LIN {X 0,Y 359.461,Z 488.763,A -85,B 0,C 180,E1 -13387.725,E2 -13387.725} C_VEL
LIN {X 0,Y 362.812,Z 518.592,A -85,B 0,C 180,E1 -13388.562,E2 -13388.562} C_VEL
LIN {X 0,Y 363.143,Z 524.633,A -85,B 0,C 180,E1 -13388.708,E2 -13388.708} C_VEL
LIN {X 0,Y 361.795,Z 606.537,A -85,B 0,C 180,E1 -13390.348,E2 -13390.348} C_VEL
LIN {X 0,Y 361.078,Z 619.618,A -85,B 0,C 180,E1 -13390.825,E2 -13390.825} C_VEL
LIN {X 0,Y 360.35,Z 632.194,A -85,B 0,C 180,E1 -13391.522,E2 -13391.522} C_VEL
LIN {X 0,Y 359.408,Z 643.388,A -85,B 0,C 180,E1 -13392.356,E2 -13392.356} C_VEL
LIN {X 0,Y 358.272,Z 654.913,A -85,B 0,C 180,E1 -13393.475,E2 -13393.475} C_VEL
LIN {X 0,Y 357.239,Z 665.304,A -85,B 0,C 180,E1 -13394.749,E2 -13394.749} C_VEL
LIN {X 0,Y 356.357,Z 673.723,A -85,B 0,C 180,E1 -13396.019,E2 -13396.019} C_VEL
LIN {X 0,Y 355.447,Z 681.49,A -85,B 0,C 180,E1 -13397.438,E2 -13397.438} C_VEL
LIN {X 0,Y 354.634,Z 689.051,A -85,B 0,C 180,E1 -13399.148,E2 -13399.148} C_VEL
LIN {X 0,Y 354.06,Z 695.119,A -85,B 0,C 180,E1 -13400.863,E2 -13400.863} C_VEL
LIN {X 0,Y 353.628,Z 699.908,A -85,B 0,C 180,E1 -13402.578,E2 -13402.578} C_VEL
LIN {X 0,Y 353.416,Z 703.562,A -85,B 0,C 180,E1 -13404.293,E2 -13404.293} C_VEL
LIN {X 0,Y 353.372,Z 705.445,A -85,B 0,C 180,E1 -13405.437,E2 -13405.437} C_VEL
LIN {X 0,Y 353.285,Z 706.865,A -85,B 0,C 180,E1 -13406.578,E2 -13406.578} C_VEL
LIN {X 0,Y 353.239,Z 708.477,A -85,B 0,C 180,E1 -13408.86,E2 -13408.86} C_VEL
LIN {X 0,Y 353.281,Z 708.695,A -85,B 0,C 180,E1 -13410,E2 -13410} C_VEL
LIN {X 0,Y 353.285,Z 708.473,A -85,B 0,C 180,E1 -13411.14,E2 -13411.14} C_VEL
LIN {X 0,Y 353.291,Z 706.855,A -85,B 0,C 180,E1 -13413.421,E2 -13413.421} C_VEL
LIN {X 0,Y 353.381,Z 705.429,A -85,B 0,C 180,E1 -13414.563,E2 -13414.563} C_VEL
LIN {X 0,Y 353.476,Z 702.599,A -85,B 0,C 180,E1 -13416.212,E2 -13416.212} C_VEL
LIN {X 0,Y 353.734,Z 698.435,A -85,B 0,C 180,E1 -13417.994,E2 -13417.994} C_VEL
LIN {X 0,Y 354.314,Z 692.219,A -85,B 0,C 180,E1 -13419.995,E2 -13419.995} C_VEL
LIN {X 0,Y 354.986,Z 685.433,A -85,B 0,C 180,E1 -13421.708,E2 -13421.708} C_VEL
LIN {X 0,Y 355.811,Z 678.485,A -85,B 0,C 180,E1 -13423.129,E2 -13423.129} C_VEL
LIN {X 0,Y 356.713,Z 670.085,A -85,B 0,C 180,E1 -13424.549,E2 -13424.549} C_VEL
LIN {X 0,Y 357.781,Z 659.681,A -85,B 0,C 180,E1 -13425.962,E2 -13425.962} C_VEL
LIN {X 0,Y 358.816,Z 649.368,A -85,B 0,C 180,E1 -13427.086,E2 -13427.086} C_VEL
LIN {X 0,Y 359.843,Z 638.003,A -85,B 0,C 180,E1 -13428.062,E2 -13428.062} C_VEL
LIN {X 0,Y 360.766,Z 624.933,A -85,B 0,C 180,E1 -13428.897,E2 -13428.897} C_VEL
LIN {X 0,Y 361.503,Z 612.616,A -85,B 0,C 180,E1 -13429.447,E2 -13429.447} C_VEL
LIN {X 0,Y 361.878,Z 602.647,A -85,B 0,C 180,E1 -13429.758,E2 -13429.758} C_VEL
LIN {X 0,Y 363.518,Z 587.437,A -85,B 0,C 180,E1 -13430.587,E2 -13430.587} C_VEL
LIN {X 0,Y 364.531,Z 572.35,A -85,B 0,C 180,E1 -13431.155,E2 -13431.155} C_VEL
LIN {X 0,Y 366.818,Z 522.316,A -85,B 0,C 180,E1 -13432.636,E2 -13432.636} C_VEL
LIN {X 0,Y 365.737,Z 500.479,A -85,B 0,C 180,E1 -13433.543,E2 -13433.543} C_VEL
LIN {X 0,Y 363.696,Z 482.777,A -85,B 0,C 180,E1 -13434.452,E2 -13434.452} C_VEL
LIN {X 0,Y 360.558,Z 464.171,A -85,B 0,C 180,E1 -13435.599,E2 -13435.599} C_VEL
LIN {X 0,Y 359.9,Z 460.319,A -85,B 0,C 180,E1 -13435.889,E2 -13435.889} C_VEL
LIN {X 0,Y 362.247,Z 444.845,A -85,B 0,C 180,E1 -13439.014,E2 -13439.014} C_VEL
LIN {X 0,Y 363.495,Z 437.862,A -85,B 0,C 180,E1 -13440.5,E2 -13440.5} C_VEL
LIN {X 0,Y 362.465,Z 431.346,A -85,B 0,C 180,E1 -13442.222,E2 -13442.222} C_VEL
LIN {X 0,Y 360.838,Z 424.073,A -85,B 0,C 180,E1 -13444.391,E2 -13444.391} C_VEL
LIN {X 0,Y 358.871,Z 416.962,A -85,B 0,C 180,E1 -13446.843,E2 -13446.843} C_VEL
LIN {X 0,Y 356.686,Z 409.94,A -85,B 0,C 180,E1 -13449.786,E2 -13449.786} C_VEL
LIN {X 0,Y 354.81,Z 404.374,A -85,B 0,C 180,E1 -13452.814,E2 -13452.814} C_VEL
LIN {X 0,Y 354.763,Z 404.295,A -85,B 0,C 180,E1 -13456.103,E2 -13456.103} C_VEL
LIN {X 0,Y 354.765,Z 404.295,A -85,B 0,C 180,E1 -13459.176,E2 -13459.176} C_VEL
LIN {X 0,Y 354.801,Z 404.288,A -85,B 0,C 180,E1 -13462.404,E2 -13462.404} C_VEL
LIN {X 0,Y 354.813,Z 404.29,A -85,B 0,C 180,E1 -13464.941,E2 -13464.941} C_VEL
LIN {X 0,Y 354.795,Z 404.292,A -85,B 0,C 180,E1 -13468.405,E2 -13468.405} C_VEL
LIN {X 0,Y 354.804,Z 404.289,A -85,B 0,C 180,E1 -13471.615,E2 -13471.615} C_VEL
LIN {X 0,Y 354.878,Z 404.452,A -85,B 0,C 180,E1 -13473.459,E2 -13473.459} C_VEL
LIN {X 0,Y 355.056,Z 405.311,A -85,B 0,C 180,E1 -13473.704,E2 -13473.704} C_VEL
LIN {X 0,Y 356.467,Z 407.983,A -85,B 0,C 180,E1 -13474.099,E2 -13474.099} C_VEL
LIN {X 0,Y 357.72,Z 409.436,A -85,B 0,C 180,E1 -13474.372,E2 -13474.372} C_VEL
LIN {X 0,Y 359.867,Z 412.919,A -85,B 0,C 180,E1 -13474.879,E2 -13474.879} C_VEL
LIN {X 0,Y 366.309,Z 424.138,A -85,B 0,C 180,E1 -13476.306,E2 -13476.306} C_VEL
LIN {X 0,Y 370.407,Z 432.325,A -85,B 0,C 180,E1 -13477.154,E2 -13477.154} C_VEL
LIN {X 0,Y 367.524,Z 483.674,A -85,B 0,C 180,E1 -13478.769,E2 -13478.769} C_VEL
LIN {X 0,Y 367.158,Z 500.037,A -85,B 0,C 180,E1 -13479.37,E2 -13479.37} C_VEL
LIN {X 0,Y 366.638,Z 513.137,A -85,B 0,C 180,E1 -13480.075,E2 -13480.075} C_VEL
LIN {X 0,Y 365.817,Z 525.138,A -85,B 0,C 180,E1 -13480.937,E2 -13480.937} C_VEL
LIN {X 0,Y 364.914,Z 535.852,A -85,B 0,C 180,E1 -13481.907,E2 -13481.907} C_VEL
LIN {X 0,Y 363.634,Z 546.798,A -85,B 0,C 180,E1 -13483.148,E2 -13483.148} C_VEL
LIN {X 0,Y 362.445,Z 556.55,A -85,B 0,C 180,E1 -13484.537,E2 -13484.537} C_VEL
LIN {X 0,Y 361.097,Z 565.838,A -85,B 0,C 180,E1 -13486.207,E2 -13486.207} C_VEL
LIN {X 0,Y 360.036,Z 572.192,A -85,B 0,C 180,E1 -13487.601,E2 -13487.601} C_VEL
LIN {X 0,Y 358.912,Z 578.359,A -85,B 0,C 180,E1 -13489.279,E2 -13489.279} C_VEL
LIN {X 0,Y 357.917,Z 583.167,A -85,B 0,C 180,E1 -13490.962,E2 -13490.962} C_VEL
LIN {X 0,Y 357.17,Z 586.752,A -85,B 0,C 180,E1 -13492.652,E2 -13492.652} C_VEL
LIN {X 0,Y 356.406,Z 589.291,A -85,B 0,C 180,E1 -13494.342,E2 -13494.342} C_VEL
LIN {X 0,Y 356.167,Z 590.371,A -85,B 0,C 180,E1 -13495.473,E2 -13495.473} C_VEL
LIN {X 0,Y 355.862,Z 591.054,A -85,B 0,C 180,E1 -13496.603,E2 -13496.603} C_VEL
LIN {X 0,Y 355.612,Z 591.321,A -85,B 0,C 180,E1 -13497.735,E2 -13497.735} C_VEL
LIN {X 0,Y 355.304,Z 591.132,A -85,B 0,C 180,E1 -13498.867,E2 -13498.867} C_VEL
LIN {X 0,Y 355.064,Z 590.518,A -85,B 0,C 180,E1 -13500,E2 -13500} C_VEL
LIN {X 0,Y 355.062,Z 589.461,A -85,B 0,C 180,E1 -13501.134,E2 -13501.134} C_VEL
LIN {X 0,Y 354.997,Z 587.96,A -85,B 0,C 180,E1 -13502.269,E2 -13502.269} C_VEL
LIN {X 0,Y 354.982,Z 584.874,A -85,B 0,C 180,E1 -13503.973,E2 -13503.973} C_VEL
LIN {X 0,Y 355.19,Z 580.69,A -85,B 0,C 180,E1 -13505.678,E2 -13505.678} C_VEL
LIN {X 0,Y 355.54,Z 574.295,A -85,B 0,C 180,E1 -13507.668,E2 -13507.668} C_VEL
LIN {X 0,Y 355.933,Z 567.286,A -85,B 0,C 180,E1 -13509.375,E2 -13509.375} C_VEL
LIN {X 0,Y 356.366,Z 558.555,A -85,B 0,C 180,E1 -13511.086,E2 -13511.086} C_VEL
LIN {X 0,Y 356.866,Z 549.666,A -85,B 0,C 180,E1 -13512.511,E2 -13512.511} C_VEL
LIN {X 0,Y 357.419,Z 538.714,A -85,B 0,C 180,E1 -13513.938,E2 -13513.938} C_VEL
LIN {X 0,Y 358.013,Z 527.922,A -85,B 0,C 180,E1 -13515.076,E2 -13515.076} C_VEL
LIN {X 0,Y 358.444,Z 515.746,A -85,B 0,C 180,E1 -13516.107,E2 -13516.107} C_VEL
LIN {X 0,Y 358.803,Z 502.919,A -85,B 0,C 180,E1 -13516.939,E2 -13516.939} C_VEL
LIN {X 0,Y 359.093,Z 490.116,A -85,B 0,C 180,E1 -13517.549,E2 -13517.549} C_VEL
LIN {X 0,Y 359.22,Z 473.341,A -85,B 0,C 180,E1 -13518.058,E2 -13518.058} C_VEL
LIN {X 0,Y 360.312,Z 421.7,A -85,B 0,C 180,E1 -13519.417,E2 -13519.417} C_VEL
LIN {X 0,Y 354.994,Z 405.051,A -85,B 0,C 180,E1 -13520.111,E2 -13520.111} C_VEL
LIN {X 0,Y 354.865,Z 404.333,A -85,B 0,C 180,E1 -13520.354,E2 -13520.354} C_VEL
LIN {X 0,Y 354.859,Z 404.284,A -85,B 0,C 180,E1 -13524.351,E2 -13524.351} C_VEL
LIN {X 0,Y 354.805,Z 404.274,A -85,B 0,C 180,E1 -13528.385,E2 -13528.385} C_VEL
LIN {X 0,Y 354.789,Z 404.289,A -85,B 0,C 180,E1 -13532.333,E2 -13532.333} C_VEL
LIN {X 0,Y 354.824,Z 404.285,A -85,B 0,C 180,E1 -13535.699,E2 -13535.699} C_VEL
LIN {X 0,Y 354.826,Z 404.286,A -85,B 0,C 180,E1 -13539.424,E2 -13539.424} C_VEL
LIN {X 0,Y 354.789,Z 404.287,A -85,B 0,C 180,E1 -13542.867,E2 -13542.867} C_VEL
LIN {X 0,Y 354.768,Z 404.291,A -85,B 0,C 180,E1 -13546.104,E2 -13546.104} C_VEL
LIN {X 0,Y 354.787,Z 404.294,A -85,B 0,C 180,E1 -13549.179,E2 -13549.179} C_VEL
LIN {X 0,Y 354.802,Z 404.275,A -85,B 0,C 180,E1 -13552.404,E2 -13552.404} C_VEL
LIN {X 0,Y 354.867,Z 404.473,A -85,B 0,C 180,E1 -13553.737,E2 -13553.737} C_VEL
LIN {X 0,Y 358.473,Z 416.958,A -85,B 0,C 180,E1 -13556.214,E2 -13556.214} C_VEL
LIN {X 0,Y 362.219,Z 432.037,A -85,B 0,C 180,E1 -13559.051,E2 -13559.051} C_VEL
LIN {X 0,Y 363.272,Z 437.662,A -85,B 0,C 180,E1 -13560.054,E2 -13560.054} C_VEL
LIN {X 0,Y 361.925,Z 456.618,A -85,B 0,C 180,E1 -13563.022,E2 -13563.022} C_VEL
LIN {X 0,Y 360.281,Z 480.837,A -85,B 0,C 180,E1 -13566.66,E2 -13566.66} C_VEL
LIN {X 0,Y 359.891,Z 488.076,A -85,B 0,C 180,E1 -13567.657,E2 -13567.657} C_VEL
LIN {X 0,Y 363.691,Z 514.331,A -85,B 0,C 180,E1 -13568.46,E2 -13568.46} C_VEL
LIN {X 0,Y 362.716,Z 576.614,A -85,B 0,C 180,E1 -13569.699,E2 -13569.699} C_VEL
LIN {X 0,Y 362.221,Z 601.278,A -85,B 0,C 180,E1 -13570.225,E2 -13570.225} C_VEL
LIN {X 0,Y 361.585,Z 613.984,A -85,B 0,C 180,E1 -13570.706,E2 -13570.706} C_VEL
LIN {X 0,Y 360.763,Z 627.4,A -85,B 0,C 180,E1 -13571.471,E2 -13571.471} C_VEL
LIN {X 0,Y 359.697,Z 639.089,A -85,B 0,C 180,E1 -13572.371,E2 -13572.371} C_VEL
LIN {X 0,Y 358.606,Z 650.259,A -85,B 0,C 180,E1 -13573.491,E2 -13573.491} C_VEL
LIN {X 0,Y 357.682,Z 660.097,A -85,B 0,C 180,E1 -13574.726,E2 -13574.726} C_VEL
LIN {X 0,Y 356.669,Z 668.662,A -85,B 0,C 180,E1 -13576.032,E2 -13576.032} C_VEL
LIN {X 0,Y 355.529,Z 677.663,A -85,B 0,C 180,E1 -13577.731,E2 -13577.731} C_VEL
LIN {X 0,Y 354.758,Z 684.885,A -85,B 0,C 180,E1 -13579.441,E2 -13579.441} C_VEL
LIN {X 0,Y 354.025,Z 691.514,A -85,B 0,C 180,E1 -13581.438,E2 -13581.438} C_VEL
LIN {X 0,Y 353.666,Z 695.868,A -85,B 0,C 180,E1 -13583.152,E2 -13583.152} C_VEL
LIN {X 0,Y 353.479,Z 698.16,A -85,B 0,C 180,E1 -13584.295,E2 -13584.295} C_VEL
LIN {X 0,Y 353.366,Z 700.029,A -85,B 0,C 180,E1 -13585.437,E2 -13585.437} C_VEL
LIN {X 0,Y 353.244,Z 701.457,A -85,B 0,C 180,E1 -13586.578,E2 -13586.578} C_VEL
LIN {X 0,Y 353.158,Z 703.075,A -85,B 0,C 180,E1 -13588.86,E2 -13588.86} C_VEL
LIN {X 0,Y 353.175,Z 703.31,A -85,B 0,C 180,E1 -13590,E2 -13590} C_VEL
LIN {X 0,Y 353.158,Z 703.117,A -85,B 0,C 180,E1 -13591.14,E2 -13591.14} C_VEL
LIN {X 0,Y 353.243,Z 701.554,A -85,B 0,C 180,E1 -13593.422,E2 -13593.422} C_VEL
LIN {X 0,Y 353.36,Z 700.18,A -85,B 0,C 180,E1 -13594.563,E2 -13594.563} C_VEL
LIN {X 0,Y 353.525,Z 697.282,A -85,B 0,C 180,E1 -13596.283,E2 -13596.283} C_VEL
LIN {X 0,Y 353.823,Z 693.372,A -85,B 0,C 180,E1 -13597.993,E2 -13597.993} C_VEL
LIN {X 0,Y 354.368,Z 688.291,A -85,B 0,C 180,E1 -13599.705,E2 -13599.705} C_VEL
LIN {X 0,Y 355.088,Z 681.888,A -85,B 0,C 180,E1 -13601.416,E2 -13601.416} C_VEL
LIN {X 0,Y 355.944,Z 674.557,A -85,B 0,C 180,E1 -13603,E2 -13603} C_VEL
LIN {X 0,Y 355.766,Z 670.779,A -85,B 0,C 180,E1 -13603.732,E2 -13603.732} C_VEL
LIN {X 0,Y 353.689,Z 664.355,A -85,B 0,C 180,E1 -13604.912,E2 -13604.912} C_VEL
LIN {X 0,Y 351.651,Z 657.479,A -85,B 0,C 180,E1 -13606.029,E2 -13606.029} C_VEL
LIN {X 0,Y 351.516,Z 652.894,A -85,B 0,C 180,E1 -13606.642,E2 -13606.642} C_VEL
LIN {X 0,Y 352.757,Z 641.711,A -85,B 0,C 180,E1 -13607.838,E2 -13607.838} C_VEL
LIN {X 0,Y 353.851,Z 629.822,A -85,B 0,C 180,E1 -13608.83,E2 -13608.83} C_VEL
LIN {X 0,Y 354.693,Z 617.392,A -85,B 0,C 180,E1 -13609.61,E2 -13609.61} C_VEL
LIN {X 0,Y 355.48,Z 604.249,A -85,B 0,C 180,E1 -13610.167,E2 -13610.167} C_VEL
LIN {X 0,Y 355.953,Z 590.394,A -85,B 0,C 180,E1 -13610.516,E2 -13610.516} C_VEL
LIN {X 0,Y 357.122,Z 514.751,A -85,B 0,C 180,E1 -13612.052,E2 -13612.052} C_VEL
LIN {X 0,Y 353.268,Z 487.892,A -85,B 0,C 180,E1 -13612.904,E2 -13612.904} C_VEL
LIN {X 0,Y 354.289,Z 470.851,A -85,B 0,C 180,E1 -13615.403,E2 -13615.403} C_VEL
LIN {X 0,Y 356.179,Z 446.213,A -85,B 0,C 180,E1 -13619.233,E2 -13619.233} C_VEL
LIN {X 0,Y 356.668,Z 440.12,A -85,B 0,C 180,E1 -13620.201,E2 -13620.201} C_VEL
LIN {X 0,Y 354.578,Z 429.7,A -85,B 0,C 180,E1 -13622.125,E2 -13622.125} C_VEL
LIN {X 0,Y 350.938,Z 415.804,A -85,B 0,C 180,E1 -13624.807,E2 -13624.807} C_VEL
LIN {X 0,Y 347.815,Z 405.367,A -85,B 0,C 180,E1 -13626.938,E2 -13626.938} C_VEL
LIN {X 0,Y 347.699,Z 405.157,A -85,B 0,C 180,E1 -13630.302,E2 -13630.302} C_VEL
LIN {X 0,Y 347.723,Z 405.159,A -85,B 0,C 180,E1 -13633.409,E2 -13633.409} C_VEL
LIN {X 0,Y 347.727,Z 405.168,A -85,B 0,C 180,E1 -13636.687,E2 -13636.687} C_VEL
LIN {X 0,Y 347.703,Z 405.174,A -85,B 0,C 180,E1 -13640.182,E2 -13640.182} C_VEL
LIN {X 0,Y 347.757,Z 405.157,A -85,B 0,C 180,E1 -13642.678,E2 -13642.678} C_VEL
LIN {X 0,Y 347.751,Z 405.158,A -85,B 0,C 180,E1 -13645.956,E2 -13645.956} C_VEL
LIN {X 0,Y 347.741,Z 405.167,A -85,B 0,C 180,E1 -13649.651,E2 -13649.651} C_VEL
LIN {X 0,Y 347.743,Z 405.172,A -85,B 0,C 180,E1 -13653.6,E2 -13653.6} C_VEL
LIN {X 0,Y 347.766,Z 405.15,A -85,B 0,C 180,E1 -13656.16,E2 -13656.16} C_VEL
LIN {X 0,Y 347.783,Z 405.162,A -85,B 0,C 180,E1 -13659.907,E2 -13659.907} C_VEL
LIN {X 0,Y 347.801,Z 405.15,A -85,B 0,C 180,E1 -13663.567,E2 -13663.567} C_VEL
LIN {X 0,Y 347.888,Z 405.141,A -85,B 0,C 180,E1 -13667.16,E2 -13667.16} C_VEL
LIN {X 0,Y 347.937,Z 405.139,A -85,B 0,C 180,E1 -13670.701,E2 -13670.701} C_VEL
LIN {X 0,Y 348.04,Z 405.116,A -85,B 0,C 180,E1 -13674.205,E2 -13674.205} C_VEL
LIN {X 0,Y 348.19,Z 405.107,A -85,B 0,C 180,E1 -13677.686,E2 -13677.686} C_VEL
LIN {X 0,Y 348.119,Z 405.109,A -85,B 0,C 180,E1 -13681.157,E2 -13681.157} C_VEL
LIN {X 0,Y 348.185,Z 405.089,A -85,B 0,C 180,E1 -13682.314,E2 -13682.314} C_VEL
LIN {X 0,Y 348.058,Z 405.127,A -85,B 0,C 180,E1 -13686.959,E2 -13686.959} C_VEL
LIN {X 0,Y 347.894,Z 405.132,A -85,B 0,C 180,E1 -13690.475,E2 -13690.475} C_VEL
LIN {X 0,Y 347.859,Z 405.15,A -85,B 0,C 180,E1 -13694.122,E2 -13694.122} C_VEL
LIN {X 0,Y 347.79,Z 405.155,A -85,B 0,C 180,E1 -13698.238,E2 -13698.238} C_VEL
LIN {X 0,Y 347.766,Z 405.156,A -85,B 0,C 180,E1 -13701.624,E2 -13701.624} C_VEL
LIN {X 0,Y 347.741,Z 405.164,A -85,B 0,C 180,E1 -13705.114,E2 -13705.114} C_VEL
LIN {X 0,Y 347.731,Z 405.161,A -85,B 0,C 180,E1 -13707.701,E2 -13707.701} C_VEL
LIN {X 0,Y 347.741,Z 405.162,A -85,B 0,C 180,E1 -13710.349,E2 -13710.349} C_VEL
LIN {X 0,Y 347.75,Z 405.154,A -85,B 0,C 180,E1 -13714.043,E2 -13714.043} C_VEL
LIN {X 0,Y 347.756,Z 405.168,A -85,B 0,C 180,E1 -13717.322,E2 -13717.322} C_VEL
LIN {X 0,Y 347.697,Z 405.133,A -85,B 0,C 180,E1 -13720.302,E2 -13720.302} C_VEL
LIN {X 0,Y 347.722,Z 405.148,A -85,B 0,C 180,E1 -13723.408,E2 -13723.408} C_VEL
LIN {X 0,Y 347.724,Z 405.164,A -85,B 0,C 180,E1 -13726.687,E2 -13726.687} C_VEL
LIN {X 0,Y 347.702,Z 405.145,A -85,B 0,C 180,E1 -13730.182,E2 -13730.182} C_VEL
LIN {X 0,Y 347.755,Z 405.168,A -85,B 0,C 180,E1 -13732.678,E2 -13732.678} C_VEL
LIN {X 0,Y 347.84,Z 405.386,A -85,B 0,C 180,E1 -13734.974,E2 -13734.974} C_VEL
LIN {X 0,Y 351.815,Z 423.417,A -85,B 0,C 180,E1 -13738.709,E2 -13738.709} C_VEL
LIN {X 0,Y 353.402,Z 430.82,A -85,B 0,C 180,E1 -13740.187,E2 -13740.187} C_VEL
LIN {X 0,Y 353.222,Z 435.729,A -85,B 0,C 180,E1 -13741.1,E2 -13741.1} C_VEL
LIN {X 0,Y 350.983,Z 459.339,A -85,B 0,C 180,E1 -13745.37,E2 -13745.37} C_VEL
LIN {X 0,Y 352.006,Z 474.914,A -85,B 0,C 180,E1 -13746.387,E2 -13746.387} C_VEL
LIN {X 0,Y 352.822,Z 488.798,A -85,B 0,C 180,E1 -13747.281,E2 -13747.281} C_VEL
LIN {X 0,Y 356.443,Z 521.377,A -85,B 0,C 180,E1 -13748.217,E2 -13748.217} C_VEL
LIN {X 0,Y 355.687,Z 575.748,A -85,B 0,C 180,E1 -13749.317,E2 -13749.317} C_VEL
LIN {X 0,Y 355.114,Z 606.569,A -85,B 0,C 180,E1 -13749.963,E2 -13749.963} C_VEL
LIN {X 0,Y 354.386,Z 619.613,A -85,B 0,C 180,E1 -13750.448,E2 -13750.448} C_VEL
LIN {X 0,Y 353.618,Z 632.173,A -85,B 0,C 180,E1 -13751.158,E2 -13751.158} C_VEL
LIN {X 0,Y 352.65,Z 643.356,A -85,B 0,C 180,E1 -13752.007,E2 -13752.007} C_VEL
LIN {X 0,Y 351.445,Z 654.875,A -85,B 0,C 180,E1 -13753.144,E2 -13753.144} C_VEL
LIN {X 0,Y 350.3,Z 665.989,A -85,B 0,C 180,E1 -13754.543,E2 -13754.543} C_VEL
LIN {X 0,Y 349.271,Z 675.329,A -85,B 0,C 180,E1 -13756.027,E2 -13756.027} C_VEL
LIN {X 0,Y 348.164,Z 684.141,A -85,B 0,C 180,E1 -13757.763,E2 -13757.763} C_VEL
LIN {X 0,Y 347.381,Z 691.2,A -85,B 0,C 180,E1 -13759.509,E2 -13759.509} C_VEL
LIN {X 0,Y 346.836,Z 696.808,A -85,B 0,C 180,E1 -13761.258,E2 -13761.258} C_VEL
LIN {X 0,Y 346.444,Z 701.198,A -85,B 0,C 180,E1 -13763.009,E2 -13763.009} C_VEL
LIN {X 0,Y 346.338,Z 703.51,A -85,B 0,C 180,E1 -13764.176,E2 -13764.176} C_VEL
LIN {X 0,Y 346.286,Z 705.392,A -85,B 0,C 180,E1 -13765.343,E2 -13765.343} C_VEL
LIN {X 0,Y 346.208,Z 706.811,A -85,B 0,C 180,E1 -13766.508,E2 -13766.508} C_VEL
LIN {X 0,Y 346.139,Z 708.424,A -85,B 0,C 180,E1 -13768.836,E2 -13768.836} C_VEL
LIN {X 0,Y 346.181,Z 708.641,A -85,B 0,C 180,E1 -13770,E2 -13770} C_VEL
LIN {X 0,Y 346.183,Z 708.419,A -85,B 0,C 180,E1 -13771.163,E2 -13771.163} C_VEL
LIN {X 0,Y 346.214,Z 706.801,A -85,B 0,C 180,E1 -13773.491,E2 -13773.491} C_VEL
LIN {X 0,Y 346.295,Z 705.375,A -85,B 0,C 180,E1 -13774.656,E2 -13774.656} C_VEL
LIN {X 0,Y 346.401,Z 702.799,A -85,B 0,C 180,E1 -13776.202,E2 -13776.202} C_VEL
LIN {X 0,Y 346.678,Z 698.38,A -85,B 0,C 180,E1 -13778.158,E2 -13778.158} C_VEL
LIN {X 0,Y 347.298,Z 692.166,A -85,B 0,C 180,E1 -13780.199,E2 -13780.199} C_VEL
LIN {X 0,Y 348.018,Z 685.381,A -85,B 0,C 180,E1 -13781.946,E2 -13781.946} C_VEL
LIN {X 0,Y 348.869,Z 678.434,A -85,B 0,C 180,E1 -13783.395,E2 -13783.395} C_VEL
LIN {X 0,Y 349.813,Z 670.035,A -85,B 0,C 180,E1 -13784.842,E2 -13784.842} C_VEL
LIN {X 0,Y 350.935,Z 659.634,A -85,B 0,C 180,E1 -13786.282,E2 -13786.282} C_VEL
LIN {X 0,Y 352.017,Z 649.324,A -85,B 0,C 180,E1 -13787.426,E2 -13787.426} C_VEL
LIN {X 0,Y 353.111,Z 637.965,A -85,B 0,C 180,E1 -13788.419,E2 -13788.419} C_VEL
LIN {X 0,Y 354.073,Z 624.904,A -85,B 0,C 180,E1 -13789.268,E2 -13789.268} C_VEL
LIN {X 0,Y 354.815,Z 612.603,A -85,B 0,C 180,E1 -13789.828,E2 -13789.828} C_VEL
LIN {X 0,Y 355.175,Z 604.546,A -85,B 0,C 180,E1 -13790.109,E2 -13790.109} C_VEL
LIN {X 0,Y 356.965,Z 589.971,A -85,B 0,C 180,E1 -13790.982,E2 -13790.982} C_VEL
LIN {X 0,Y 358.206,Z 575.233,A -85,B 0,C 180,E1 -13791.622,E2 -13791.622} C_VEL
LIN {X 0,Y 360.877,Z 523.641,A -85,B 0,C 180,E1 -13793.205,E2 -13793.205} C_VEL
LIN {X 0,Y 359.91,Z 501.776,A -85,B 0,C 180,E1 -13794.15,E2 -13794.15} C_VEL
LIN {X 0,Y 358.015,Z 484.588,A -85,B 0,C 180,E1 -13795.074,E2 -13795.074} C_VEL
LIN {X 0,Y 355.218,Z 467.047,A -85,B 0,C 180,E1 -13796.191,E2 -13796.191} C_VEL
LIN {X 0,Y 353.681,Z 458.471,A -85,B 0,C 180,E1 -13796.837,E2 -13796.837} C_VEL
LIN {X 0,Y 356.403,Z 442.572,A -85,B 0,C 180,E1 -13800.188,E2 -13800.188} C_VEL
LIN {X 0,Y 356.899,Z 439.821,A -85,B 0,C 180,E1 -13800.796,E2 -13800.796} C_VEL
LIN {X 0,Y 355.608,Z 432.185,A -85,B 0,C 180,E1 -13802.922,E2 -13802.922} C_VEL
LIN {X 0,Y 353.753,Z 424.318,A -85,B 0,C 180,E1 -13805.457,E2 -13805.457} C_VEL
LIN {X 0,Y 352.199,Z 418.863,A -85,B 0,C 180,E1 -13807.498,E2 -13807.498} C_VEL
LIN {X 0,Y 350.206,Z 412.597,A -85,B 0,C 180,E1 -13810.307,E2 -13810.307} C_VEL
LIN {X 0,Y 348.392,Z 407.393,A -85,B 0,C 180,E1 -13813.304,E2 -13813.304} C_VEL
LIN {X 0,Y 347.704,Z 405.199,A -85,B 0,C 180,E1 -13815.027,E2 -13815.027} C_VEL
LIN {X 0,Y 347.74,Z 405.167,A -85,B 0,C 180,E1 -13818.399,E2 -13818.399} C_VEL
LIN {X 0,Y 347.757,Z 405.167,A -85,B 0,C 180,E1 -13822.678,E2 -13822.678} C_VEL
LIN {X 0,Y 347.749,Z 405.166,A -85,B 0,C 180,E1 -13825.956,E2 -13825.956} C_VEL
LIN {X 0,Y 347.742,Z 405.168,A -85,B 0,C 180,E1 -13829.651,E2 -13829.651} C_VEL
LIN {X 0,Y 347.797,Z 405.409,A -85,B 0,C 180,E1 -13832.223,E2 -13832.223} C_VEL
LIN {X 0,Y 347.973,Z 406.187,A -85,B 0,C 180,E1 -13832.441,E2 -13832.441} C_VEL
LIN {X 0,Y 349.437,Z 408.915,A -85,B 0,C 180,E1 -13832.889,E2 -13832.889} C_VEL
LIN {X 0,Y 351.057,Z 410.737,A -85,B 0,C 180,E1 -13833.29,E2 -13833.29} C_VEL
LIN {X 0,Y 353.011,Z 413.918,A -85,B 0,C 180,E1 -13833.818,E2 -13833.818} C_VEL
LIN {X 0,Y 358.572,Z 423.002,A -85,B 0,C 180,E1 -13835.153,E2 -13835.153} C_VEL
LIN {X 0,Y 364.152,Z 433.748,A -85,B 0,C 180,E1 -13836.426,E2 -13836.426} C_VEL
LIN {X 0,Y 364.737,Z 435.343,A -85,B 0,C 180,E1 -13836.567,E2 -13836.567} C_VEL
LIN {X 0,Y 361.707,Z 483.693,A -85,B 0,C 180,E1 -13838.123,E2 -13838.123} C_VEL
LIN {X 0,Y 361.209,Z 501.37,A -85,B 0,C 180,E1 -13838.798,E2 -13838.798} C_VEL
LIN {X 0,Y 360.699,Z 513.766,A -85,B 0,C 180,E1 -13839.469,E2 -13839.469} C_VEL
LIN {X 0,Y 359.898,Z 524.737,A -85,B 0,C 180,E1 -13840.247,E2 -13840.247} C_VEL
LIN {X 0,Y 358.866,Z 536.261,A -85,B 0,C 180,E1 -13841.296,E2 -13841.296} C_VEL
LIN {X 0,Y 357.483,Z 547.309,A -85,B 0,C 180,E1 -13842.554,E2 -13842.554} C_VEL
LIN {X 0,Y 356.203,Z 557.181,A -85,B 0,C 180,E1 -13843.965,E2 -13843.965} C_VEL
LIN {X 0,Y 354.989,Z 565.242,A -85,B 0,C 180,E1 -13845.379,E2 -13845.379} C_VEL
LIN {X 0,Y 353.608,Z 572.804,A -85,B 0,C 180,E1 -13847.021,E2 -13847.021} C_VEL
LIN {X 0,Y 352.559,Z 578.282,A -85,B 0,C 180,E1 -13848.502,E2 -13848.502} C_VEL
LIN {X 0,Y 351.488,Z 583.348,A -85,B 0,C 180,E1 -13850.215,E2 -13850.215} C_VEL
LIN {X 0,Y 350.469,Z 587.238,A -85,B 0,C 180,E1 -13851.931,E2 -13851.931} C_VEL
LIN {X 0,Y 349.925,Z 589.217,A -85,B 0,C 180,E1 -13853.079,E2 -13853.079} C_VEL
LIN {X 0,Y 349.498,Z 590.68,A -85,B 0,C 180,E1 -13854.23,E2 -13854.23} C_VEL
LIN {X 0,Y 349.232,Z 591.682,A -85,B 0,C 180,E1 -13855.383,E2 -13855.383} C_VEL
LIN {X 0,Y 348.885,Z 592.298,A -85,B 0,C 180,E1 -13856.535,E2 -13856.535} C_VEL
LIN {X 0,Y 348.619,Z 592.461,A -85,B 0,C 180,E1 -13857.689,E2 -13857.689} C_VEL
LIN {X 0,Y 348.294,Z 592.197,A -85,B 0,C 180,E1 -13858.844,E2 -13858.844} C_VEL
LIN {X 0,Y 348.036,Z 591.518,A -85,B 0,C 180,E1 -13860,E2 -13860} C_VEL
LIN {X 0,Y 348.036,Z 590.378,A -85,B 0,C 180,E1 -13861.157,E2 -13861.157} C_VEL
LIN {X 0,Y 347.965,Z 587.843,A -85,B 0,C 180,E1 -13862.894,E2 -13862.894} C_VEL
LIN {X 0,Y 347.885,Z 584.272,A -85,B 0,C 180,E1 -13864.635,E2 -13864.635} C_VEL
LIN {X 0,Y 348.277,Z 579.533,A -85,B 0,C 180,E1 -13866.372,E2 -13866.372} C_VEL
LIN {X 0,Y 348.571,Z 573.545,A -85,B 0,C 180,E1 -13868.114,E2 -13868.114} C_VEL
LIN {X 0,Y 348.975,Z 566.105,A -85,B 0,C 180,E1 -13869.857,E2 -13869.857} C_VEL
LIN {X 0,Y 349.39,Z 558.54,A -85,B 0,C 180,E1 -13871.31,E2 -13871.31} C_VEL
LIN {X 0,Y 349.926,Z 548.358,A -85,B 0,C 180,E1 -13872.911,E2 -13872.911} C_VEL
LIN {X 0,Y 350.537,Z 536.912,A -85,B 0,C 180,E1 -13874.366,E2 -13874.366} C_VEL
LIN {X 0,Y 351.172,Z 525.512,A -85,B 0,C 180,E1 -13875.514,E2 -13875.514} C_VEL
LIN {X 0,Y 351.599,Z 512.622,A -85,B 0,C 180,E1 -13876.549,E2 -13876.549} C_VEL
LIN {X 0,Y 351.962,Z 499.83,A -85,B 0,C 180,E1 -13877.316,E2 -13877.316} C_VEL
LIN {X 0,Y 352.202,Z 486.115,A -85,B 0,C 180,E1 -13877.904,E2 -13877.904} C_VEL
LIN {X 0,Y 352.864,Z 445.943,A -85,B 0,C 180,E1 -13879,E2 -13879} C_VEL
LIN {X 0,Y 353.285,Z 422.754,A -85,B 0,C 180,E1 -13879.64,E2 -13879.64} C_VEL
LIN {X 0,Y 348.008,Z 406.168,A -85,B 0,C 180,E1 -13880.331,E2 -13880.331} C_VEL
LIN {X 0,Y 347.826,Z 405.249,A -85,B 0,C 180,E1 -13880.552,E2 -13880.552} C_VEL
LIN {X 0,Y 347.813,Z 405.162,A -85,B 0,C 180,E1 -13884.593,E2 -13884.593} C_VEL
LIN {X 0,Y 347.743,Z 405.159,A -85,B 0,C 180,E1 -13887.7,E2 -13887.7} C_VEL
LIN {X 0,Y 347.743,Z 405.163,A -85,B 0,C 180,E1 -13890.349,E2 -13890.349} C_VEL
LIN {X 0,Y 347.75,Z 405.152,A -85,B 0,C 180,E1 -13894.044,E2 -13894.044} C_VEL
LIN {X 0,Y 347.763,Z 405.16,A -85,B 0,C 180,E1 -13897.321,E2 -13897.321} C_VEL
LIN {X 0,Y 347.734,Z 405.172,A -85,B 0,C 180,E1 -13900.297,E2 -13900.297} C_VEL
LIN {X 0,Y 347.725,Z 405.172,A -85,B 0,C 180,E1 -13903.408,E2 -13903.408} C_VEL
LIN {X 0,Y 347.727,Z 405.173,A -85,B 0,C 180,E1 -13906.686,E2 -13906.686} C_VEL
LIN {X 0,Y 347.73,Z 405.159,A -85,B 0,C 180,E1 -13910.177,E2 -13910.177} C_VEL
LIN {X 0,Y 347.79,Z 405.363,A -85,B 0,C 180,E1 -13913.171,E2 -13913.171} C_VEL
LIN {X 0,Y 351.416,Z 417.393,A -85,B 0,C 180,E1 -13915.62,E2 -13915.62} C_VEL
LIN {X 0,Y 354.973,Z 431.63,A -85,B 0,C 180,E1 -13918.359,E2 -13918.359} C_VEL
LIN {X 0,Y 356.568,Z 439.347,A -85,B 0,C 180,E1 -13919.784,E2 -13919.784} C_VEL
LIN {X 0,Y 355.266,Z 457.299,A -85,B 0,C 180,E1 -13922.617,E2 -13922.617} C_VEL
LIN {X 0,Y 353.644,Z 480.117,A -85,B 0,C 180,E1 -13926.088,E2 -13926.088} C_VEL
LIN {X 0,Y 353.202,Z 488.114,A -85,B 0,C 180,E1 -13927.213,E2 -13927.213} C_VEL
LIN {X 0,Y 357.131,Z 515.394,A -85,B 0,C 180,E1 -13928.067,E2 -13928.067} C_VEL
LIN {X 0,Y 355.665,Z 598.661,A -85,B 0,C 180,E1 -13929.769,E2 -13929.769} C_VEL
LIN {X 0,Y 355.037,Z 611.718,A -85,B 0,C 180,E1 -13930.222,E2 -13930.222} C_VEL
LIN {X 0,Y 354.396,Z 623.121,A -85,B 0,C 180,E1 -13930.825,E2 -13930.825} C_VEL
LIN {X 0,Y 353.433,Z 634.124,A -85,B 0,C 180,E1 -13931.599,E2 -13931.599} C_VEL
LIN {X 0,Y 352.359,Z 645.038,A -85,B 0,C 180,E1 -13932.592,E2 -13932.592} C_VEL
LIN {X 0,Y 351.242,Z 655.794,A -85,B 0,C 180,E1 -13933.829,E2 -13933.829} C_VEL
LIN {X 0,Y 350.238,Z 665.225,A -85,B 0,C 180,E1 -13935.176,E2 -13935.176} C_VEL
LIN {X 0,Y 348.941,Z 674.928,A -85,B 0,C 180,E1 -13936.904,E2 -13936.904} C_VEL
LIN {X 0,Y 348.026,Z 682.727,A -85,B 0,C 180,E1 -13938.645,E2 -13938.645} C_VEL
LIN {X 0,Y 347.413,Z 687.998,A -85,B 0,C 180,E1 -13940.099,E2 -13940.099} C_VEL
LIN {X 0,Y 346.831,Z 693.15,A -85,B 0,C 180,E1 -13941.846,E2 -13941.846} C_VEL
LIN {X 0,Y 346.501,Z 697.248,A -85,B 0,C 180,E1 -13943.648,E2 -13943.648} C_VEL
LIN {X 0,Y 346.285,Z 700.083,A -85,B 0,C 180,E1 -13945.344,E2 -13945.344} C_VEL
LIN {X 0,Y 346.171,Z 701.511,A -85,B 0,C 180,E1 -13946.508,E2 -13946.508} C_VEL
LIN {X 0,Y 346.061,Z 703.129,A -85,B 0,C 180,E1 -13948.836,E2 -13948.836} C_VEL
LIN {X 0,Y 346.076,Z 703.364,A -85,B 0,C 180,E1 -13950,E2 -13950} C_VEL
LIN {X 0,Y 346.061,Z 703.171,A -85,B 0,C 180,E1 -13951.164,E2 -13951.164} C_VEL
LIN {X 0,Y 346.17,Z 701.607,A -85,B 0,C 180,E1 -13953.492,E2 -13953.492} C_VEL
LIN {X 0,Y 346.279,Z 700.233,A -85,B 0,C 180,E1 -13954.657,E2 -13954.657} C_VEL
LIN {X 0,Y 346.449,Z 697.588,A -85,B 0,C 180,E1 -13956.274,E2 -13956.274} C_VEL
LIN {X 0,Y 346.776,Z 693.424,A -85,B 0,C 180,E1 -13958.156,E2 -13958.156} C_VEL
LIN {X 0,Y 347.352,Z 688.342,A -85,B 0,C 180,E1 -13959.903,E2 -13959.903} C_VEL
LIN {X 0,Y 348.097,Z 681.937,A -85,B 0,C 180,E1 -13961.648,E2 -13961.648} C_VEL
LIN {X 0,Y 349.12,Z 673.98,A -85,B 0,C 180,E1 -13963.386,E2 -13963.386} C_VEL
LIN {X 0,Y 350.19,Z 665.85,A -85,B 0,C 180,E1 -13964.826,E2 -13964.826} C_VEL
LIN {X 0,Y 351.03,Z 657.532,A -85,B 0,C 180,E1 -13966.051,E2 -13966.051} C_VEL
LIN {X 0,Y 351.516,Z 652.894,A -85,B 0,C 180,E1 -13966.642,E2 -13966.642} C_VEL
LIN {X 0,Y 351.412,Z 648.185,A -85,B 0,C 180,E1 -13967.227,E2 -13967.227} C_VEL
LIN {X 0,Y 349.492,Z 640.329,A -85,B 0,C 180,E1 -13968.171,E2 -13968.171} C_VEL
LIN {X 0,Y 347.547,Z 632.07,A -85,B 0,C 180,E1 -13969.013,E2 -13969.013} C_VEL
LIN {X 0,Y 347.39,Z 626.736,A -85,B 0,C 180,E1 -13969.428,E2 -13969.428} C_VEL
LIN {X 0,Y 348.318,Z 613.853,A -85,B 0,C 180,E1 -13970.176,E2 -13970.176} C_VEL
LIN {X 0,Y 348.988,Z 600.923,A -85,B 0,C 180,E1 -13970.674,E2 -13970.674} C_VEL
LIN {X 0,Y 350.225,Z 537.89,A -85,B 0,C 180,E1 -13972.003,E2 -13972.003} C_VEL
LIN {X 0,Y 350.527,Z 515.486,A -85,B 0,C 180,E1 -13972.471,E2 -13972.471} C_VEL
LIN {X 0,Y 346.57,Z 487.86,A -85,B 0,C 180,E1 -13973.373,E2 -13973.373} C_VEL
LIN {X 0,Y 347.53,Z 472.778,A -85,B 0,C 180,E1 -13975.611,E2 -13975.611} C_VEL
LIN {X 0,Y 349.48,Z 447.819,A -85,B 0,C 180,E1 -13979.518,E2 -13979.518} C_VEL
LIN {X 0,Y 350.009,Z 441.981,A -85,B 0,C 180,E1 -13980.464,E2 -13980.464} C_VEL
LIN {X 0,Y 347.874,Z 431.55,A -85,B 0,C 180,E1 -13982.425,E2 -13982.425} C_VEL
LIN {X 0,Y 344.11,Z 417.265,A -85,B 0,C 180,E1 -13985.219,E2 -13985.219} C_VEL
LIN {X 0,Y 340.775,Z 406.267,A -85,B 0,C 180,E1 -13987.527,E2 -13987.527} C_VEL
LIN {X 0,Y 340.696,Z 406.051,A -85,B 0,C 180,E1 -13988.383,E2 -13988.383} C_VEL
LIN {X 0,Y 340.695,Z 406.047,A -85,B 0,C 180,E1 -13992.044,E2 -13992.044} C_VEL
LIN {X 0,Y 340.653,Z 406.038,A -85,B 0,C 180,E1 -13996.227,E2 -13996.227} C_VEL
LIN {X 0,Y 340.673,Z 406.047,A -85,B 0,C 180,E1 -13998.688,E2 -13998.688} C_VEL
LIN {X 0,Y 340.721,Z 406.039,A -85,B 0,C 180,E1 -14001.771,E2 -14001.771} C_VEL
LIN {X 0,Y 340.725,Z 406.037,A -85,B 0,C 180,E1 -14005.596,E2 -14005.596} C_VEL
LIN {X 0,Y 340.696,Z 406.047,A -85,B 0,C 180,E1 -14008.955,E2 -14008.955} C_VEL
LIN {X 0,Y 340.715,Z 406.042,A -85,B 0,C 180,E1 -14013.012,E2 -14013.012} C_VEL
LIN {X 0,Y 340.742,Z 406.028,A -85,B 0,C 180,E1 -14015.637,E2 -14015.637} C_VEL
LIN {X 0,Y 340.72,Z 406.046,A -85,B 0,C 180,E1 -14019.472,E2 -14019.472} C_VEL
LIN {X 0,Y 340.764,Z 406.02,A -85,B 0,C 180,E1 -14021.979,E2 -14021.979} C_VEL
LIN {X 0,Y 340.835,Z 406.03,A -85,B 0,C 180,E1 -14025.73,E2 -14025.73} C_VEL
LIN {X 0,Y 340.847,Z 406.006,A -85,B 0,C 180,E1 -14029.305,E2 -14029.305} C_VEL
LIN {X 0,Y 341.003,Z 406.005,A -85,B 0,C 180,E1 -14032.897,E2 -14032.897} C_VEL
LIN {X 0,Y 340.81,Z 406.009,A -85,B 0,C 180,E1 -14035.268,E2 -14035.268} C_VEL
LIN {X 0,Y 341.127,Z 405.986,A -85,B 0,C 180,E1 -14037.638,E2 -14037.638} C_VEL
LIN {X 0,Y 341.091,Z 405.983,A -85,B 0,C 180,E1 -14041.181,E2 -14041.181} C_VEL
LIN {X 0,Y 341.121,Z 405.968,A -85,B 0,C 180,E1 -14042.362,E2 -14042.362} C_VEL
LIN {X 0,Y 341.018,Z 406.009,A -85,B 0,C 180,E1 -14045.914,E2 -14045.914} C_VEL
LIN {X 0,Y 340.967,Z 405.998,A -85,B 0,C 180,E1 -14048.356,E2 -14048.356} C_VEL
LIN {X 0,Y 340.848,Z 406.022,A -85,B 0,C 180,E1 -14051.899,E2 -14051.899} C_VEL
LIN {X 0,Y 340.736,Z 406.024,A -85,B 0,C 180,E1 -14055.553,E2 -14055.553} C_VEL
LIN {X 0,Y 340.753,Z 406.034,A -85,B 0,C 180,E1 -14058.422,E2 -14058.422} C_VEL
LIN {X 0,Y 340.721,Z 406.03,A -85,B 0,C 180,E1 -14061.841,E2 -14061.841} C_VEL
LIN {X 0,Y 340.674,Z 406.048,A -85,B 0,C 180,E1 -14065.672,E2 -14065.672} C_VEL
LIN {X 0,Y 340.681,Z 406.032,A -85,B 0,C 180,E1 -14068.325,E2 -14068.325} C_VEL
LIN {X 0,Y 340.696,Z 406.043,A -85,B 0,C 180,E1 -14071.045,E2 -14071.045} C_VEL
LIN {X 0,Y 340.717,Z 406.033,A -85,B 0,C 180,E1 -14075.279,E2 -14075.279} C_VEL
LIN {X 0,Y 340.694,Z 406.038,A -85,B 0,C 180,E1 -14078.382,E2 -14078.382} C_VEL
LIN {X 0,Y 340.692,Z 405.999,A -85,B 0,C 180,E1 -14082.043,E2 -14082.043} C_VEL
LIN {X 0,Y 340.651,Z 406.048,A -85,B 0,C 180,E1 -14086.227,E2 -14086.227} C_VEL
LIN {X 0,Y 340.669,Z 406.01,A -85,B 0,C 180,E1 -14088.687,E2 -14088.687} C_VEL
LIN {X 0,Y 340.719,Z 406.044,A -85,B 0,C 180,E1 -14091.77,E2 -14091.77} C_VEL
LIN {X 0,Y 340.8,Z 406.251,A -85,B 0,C 180,E1 -14094.708,E2 -14094.708} C_VEL
LIN {X 0,Y 344.663,Z 423.987,A -85,B 0,C 180,E1 -14098.461,E2 -14098.461} C_VEL
LIN {X 0,Y 346.492,Z 432.57,A -85,B 0,C 180,E1 -14100.202,E2 -14100.202} C_VEL
LIN {X 0,Y 345.388,Z 444.459,A -85,B 0,C 180,E1 -14102.424,E2 -14102.424} C_VEL
LIN {X 0,Y 344.203,Z 456.865,A -85,B 0,C 180,E1 -14104.69,E2 -14104.69} C_VEL
LIN {X 0,Y 345.965,Z 485.155,A -85,B 0,C 180,E1 -14106.595,E2 -14106.595} C_VEL
LIN {X 0,Y 346.2,Z 489.111,A -85,B 0,C 180,E1 -14106.827,E2 -14106.827} C_VEL
LIN {X 0,Y 349.362,Z 517.167,A -85,B 0,C 180,E1 -14107.659,E2 -14107.659} C_VEL
LIN {X 0,Y 349.978,Z 524.863,A -85,B 0,C 180,E1 -14107.867,E2 -14107.867} C_VEL
LIN {X 0,Y 348.467,Z 606.6,A -85,B 0,C 180,E1 -14109.563,E2 -14109.563} C_VEL
LIN {X 0,Y 347.722,Z 619.607,A -85,B 0,C 180,E1 -14110.058,E2 -14110.058} C_VEL
LIN {X 0,Y 346.893,Z 632.151,A -85,B 0,C 180,E1 -14110.778,E2 -14110.778} C_VEL
LIN {X 0,Y 345.889,Z 643.324,A -85,B 0,C 180,E1 -14111.643,E2 -14111.643} C_VEL
LIN {X 0,Y 344.66,Z 654.836,A -85,B 0,C 180,E1 -14112.802,E2 -14112.802} C_VEL
LIN {X 0,Y 343.532,Z 665.16,A -85,B 0,C 180,E1 -14114.116,E2 -14114.116} C_VEL
LIN {X 0,Y 342.559,Z 673.632,A -85,B 0,C 180,E1 -14115.444,E2 -14115.444} C_VEL
LIN {X 0,Y 341.574,Z 681.394,A -85,B 0,C 180,E1 -14116.919,E2 -14116.919} C_VEL
LIN {X 0,Y 340.661,Z 688.951,A -85,B 0,C 180,E1 -14118.697,E2 -14118.697} C_VEL
LIN {X 0,Y 339.987,Z 695.017,A -85,B 0,C 180,E1 -14120.481,E2 -14120.481} C_VEL
LIN {X 0,Y 339.506,Z 699.804,A -85,B 0,C 180,E1 -14122.267,E2 -14122.267} C_VEL
LIN {X 0,Y 339.259,Z 703.457,A -85,B 0,C 180,E1 -14124.055,E2 -14124.055} C_VEL
LIN {X 0,Y 339.204,Z 705.339,A -85,B 0,C 180,E1 -14125.246,E2 -14125.246} C_VEL
LIN {X 0,Y 339.133,Z 706.758,A -85,B 0,C 180,E1 -14126.435,E2 -14126.435} C_VEL
LIN {X 0,Y 339.041,Z 708.37,A -85,B 0,C 180,E1 -14128.812,E2 -14128.812} C_VEL
LIN {X 0,Y 339.081,Z 708.587,A -85,B 0,C 180,E1 -14130,E2 -14130} C_VEL
LIN {X 0,Y 339.082,Z 708.365,A -85,B 0,C 180,E1 -14131.187,E2 -14131.187} C_VEL
LIN {X 0,Y 339.139,Z 706.746,A -85,B 0,C 180,E1 -14133.564,E2 -14133.564} C_VEL
LIN {X 0,Y 339.213,Z 705.321,A -85,B 0,C 180,E1 -14134.754,E2 -14134.754} C_VEL
LIN {X 0,Y 339.291,Z 703.089,A -85,B 0,C 180,E1 -14136.139,E2 -14136.139} C_VEL
LIN {X 0,Y 339.625,Z 698.326,A -85,B 0,C 180,E1 -14138.329,E2 -14138.329} C_VEL
LIN {X 0,Y 340.288,Z 692.112,A -85,B 0,C 180,E1 -14140.411,E2 -14140.411} C_VEL
LIN {X 0,Y 341.06,Z 685.328,A -85,B 0,C 180,E1 -14142.193,E2 -14142.193} C_VEL
LIN {X 0,Y 341.936,Z 678.383,A -85,B 0,C 180,E1 -14143.672,E2 -14143.672} C_VEL
LIN {X 0,Y 342.931,Z 669.985,A -85,B 0,C 180,E1 -14145.147,E2 -14145.147} C_VEL
LIN {X 0,Y 344.098,Z 659.587,A -85,B 0,C 180,E1 -14146.615,E2 -14146.615} C_VEL
LIN {X 0,Y 345.245,Z 649.28,A -85,B 0,C 180,E1 -14147.779,E2 -14147.779} C_VEL
LIN {X 0,Y 346.386,Z 637.926,A -85,B 0,C 180,E1 -14148.79,E2 -14148.79} C_VEL
LIN {X 0,Y 347.279,Z 626.153,A -85,B 0,C 180,E1 -14149.583,E2 -14149.583} C_VEL
LIN {X 0,Y 348.123,Z 613.481,A -85,B 0,C 180,E1 -14150.187,E2 -14150.187} C_VEL
LIN {X 0,Y 348.457,Z 606.891,A -85,B 0,C 180,E1 -14150.437,E2 -14150.437} C_VEL
LIN {X 0,Y 350.403,Z 592.451,A -85,B 0,C 180,E1 -14151.394,E2 -14151.394} C_VEL
LIN {X 0,Y 351.849,Z 578.686,A -85,B 0,C 180,E1 -14152.072,E2 -14152.072} C_VEL
LIN {X 0,Y 353.167,Z 557.185,A -85,B 0,C 180,E1 -14152.793,E2 -14152.793} C_VEL
LIN {X 0,Y 354.98,Z 523.736,A -85,B 0,C 180,E1 -14153.862,E2 -14153.862} C_VEL
LIN {X 0,Y 354.216,Z 503.49,A -85,B 0,C 180,E1 -14154.771,E2 -14154.771} C_VEL
LIN {X 0,Y 352.534,Z 486.904,A -85,B 0,C 180,E1 -14155.695,E2 -14155.695} C_VEL
LIN {X 0,Y 350.101,Z 470.268,A -85,B 0,C 180,E1 -14156.795,E2 -14156.795} C_VEL
LIN {X 0,Y 347.591,Z 456.61,A -85,B 0,C 180,E1 -14157.877,E2 -14157.877} C_VEL
LIN {X 0,Y 350.111,Z 443.17,A -85,B 0,C 180,E1 -14160.789,E2 -14160.789} C_VEL
LIN {X 0,Y 350.185,Z 440.557,A -85,B 0,C 180,E1 -14161.453,E2 -14161.453} C_VEL
LIN {X 0,Y 348.666,Z 432.558,A -85,B 0,C 180,E1 -14163.844,E2 -14163.844} C_VEL
LIN {X 0,Y 346.875,Z 425.365,A -85,B 0,C 180,E1 -14166.344,E2 -14166.344} C_VEL
LIN {X 0,Y 344.819,Z 418.457,A -85,B 0,C 180,E1 -14169.24,E2 -14169.24} C_VEL
LIN {X 0,Y 343.516,Z 414.428,A -85,B 0,C 180,E1 -14171.295,E2 -14171.295} C_VEL
LIN {X 0,Y 341.978,Z 410.178,A -85,B 0,C 180,E1 -14174.004,E2 -14174.004} C_VEL
LIN {X 0,Y 340.771,Z 406.622,A -85,B 0,C 180,E1 -14177.11,E2 -14177.11} C_VEL
LIN {X 0,Y 340.71,Z 406.062,A -85,B 0,C 180,E1 -14177.953,E2 -14177.953} C_VEL
LIN {X 0,Y 340.719,Z 406.041,A -85,B 0,C 180,E1 -14181.771,E2 -14181.771} C_VEL
LIN {X 0,Y 340.724,Z 406.04,A -85,B 0,C 180,E1 -14185.595,E2 -14185.595} C_VEL
LIN {X 0,Y 340.696,Z 406.045,A -85,B 0,C 180,E1 -14188.955,E2 -14188.955} C_VEL
LIN {X 0,Y 340.75,Z 406.328,A -85,B 0,C 180,E1 -14190.752,E2 -14190.752} C_VEL
LIN {X 0,Y 340.918,Z 407.022,A -85,B 0,C 180,E1 -14190.978,E2 -14190.978} C_VEL
LIN {X 0,Y 342.359,Z 409.755,A -85,B 0,C 180,E1 -14191.513,E2 -14191.513} C_VEL
LIN {X 0,Y 344.032,Z 411.49,A -85,B 0,C 180,E1 -14191.975,E2 -14191.975} C_VEL
LIN {X 0,Y 345.814,Z 414.568,A -85,B 0,C 180,E1 -14192.513,E2 -14192.513} C_VEL
LIN {X 0,Y 347.268,Z 416.415,A -85,B 0,C 180,E1 -14192.895,E2 -14192.895} C_VEL
LIN {X 0,Y 351.98,Z 423.994,A -85,B 0,C 180,E1 -14194.143,E2 -14194.143} C_VEL
LIN {X 0,Y 357.383,Z 433.893,A -85,B 0,C 180,E1 -14195.473,E2 -14195.473} C_VEL
LIN {X 0,Y 359.207,Z 437.935,A -85,B 0,C 180,E1 -14195.918,E2 -14195.918} C_VEL
LIN {X 0,Y 356.012,Z 483.537,A -85,B 0,C 180,E1 -14197.436,E2 -14197.436} C_VEL
LIN {X 0,Y 355.424,Z 501.843,A -85,B 0,C 180,E1 -14198.139,E2 -14198.139} C_VEL
LIN {X 0,Y 354.756,Z 515.573,A -85,B 0,C 180,E1 -14198.903,E2 -14198.903} C_VEL
LIN {X 0,Y 353.842,Z 526.916,A -85,B 0,C 180,E1 -14199.749,E2 -14199.749} C_VEL
LIN {X 0,Y 352.744,Z 538.22,A -85,B 0,C 180,E1 -14200.807,E2 -14200.807} C_VEL
LIN {X 0,Y 351.271,Z 549.136,A -85,B 0,C 180,E1 -14202.085,E2 -14202.085} C_VEL
LIN {X 0,Y 349.751,Z 559.714,A -85,B 0,C 180,E1 -14203.661,E2 -14203.661} C_VEL
LIN {X 0,Y 348.191,Z 568.83,A -85,B 0,C 180,E1 -14205.386,E2 -14205.386} C_VEL
LIN {X 0,Y 346.73,Z 576.199,A -85,B 0,C 180,E1 -14207.117,E2 -14207.117} C_VEL
LIN {X 0,Y 345.422,Z 581.975,A -85,B 0,C 180,E1 -14208.855,E2 -14208.855} C_VEL
LIN {X 0,Y 344.296,Z 586.454,A -85,B 0,C 180,E1 -14210.601,E2 -14210.601} C_VEL
LIN {X 0,Y 343.635,Z 588.804,A -85,B 0,C 180,E1 -14211.769,E2 -14211.769} C_VEL
LIN {X 0,Y 343.032,Z 590.688,A -85,B 0,C 180,E1 -14212.939,E2 -14212.939} C_VEL
LIN {X 0,Y 342.584,Z 592.067,A -85,B 0,C 180,E1 -14214.113,E2 -14214.113} C_VEL
LIN {X 0,Y 342.291,Z 593.007,A -85,B 0,C 180,E1 -14215.289,E2 -14215.289} C_VEL
LIN {X 0,Y 341.926,Z 593.54,A -85,B 0,C 180,E1 -14216.465,E2 -14216.465} C_VEL
LIN {X 0,Y 341.624,Z 593.605,A -85,B 0,C 180,E1 -14217.642,E2 -14217.642} C_VEL
LIN {X 0,Y 341.303,Z 593.268,A -85,B 0,C 180,E1 -14218.82,E2 -14218.82} C_VEL
LIN {X 0,Y 341.008,Z 592.514,A -85,B 0,C 180,E1 -14220,E2 -14220} C_VEL
LIN {X 0,Y 341.01,Z 591.259,A -85,B 0,C 180,E1 -14221.181,E2 -14221.181} C_VEL
LIN {X 0,Y 340.927,Z 588.598,A -85,B 0,C 180,E1 -14222.954,E2 -14222.954} C_VEL
LIN {X 0,Y 340.856,Z 584.887,A -85,B 0,C 180,E1 -14224.731,E2 -14224.731} C_VEL
LIN {X 0,Y 341.235,Z 579.996,A -85,B 0,C 180,E1 -14226.504,E2 -14226.504} C_VEL
LIN {X 0,Y 341.557,Z 573.835,A -85,B 0,C 180,E1 -14228.281,E2 -14228.281} C_VEL
LIN {X 0,Y 341.968,Z 566.178,A -85,B 0,C 180,E1 -14230.061,E2 -14230.061} C_VEL
LIN {X 0,Y 342.503,Z 556.622,A -85,B 0,C 180,E1 -14231.841,E2 -14231.841} C_VEL
LIN {X 0,Y 343.047,Z 546.844,A -85,B 0,C 180,E1 -14233.325,E2 -14233.325} C_VEL
LIN {X 0,Y 343.587,Z 535.988,A -85,B 0,C 180,E1 -14234.663,E2 -14234.663} C_VEL
LIN {X 0,Y 344.176,Z 524.775,A -85,B 0,C 180,E1 -14235.784,E2 -14235.784} C_VEL
LIN {X 0,Y 344.616,Z 512.743,A -85,B 0,C 180,E1 -14236.742,E2 -14236.742} C_VEL
LIN {X 0,Y 344.97,Z 498.313,A -85,B 0,C 180,E1 -14237.602,E2 -14237.602} C_VEL
LIN {X 0,Y 345.236,Z 484.393,A -85,B 0,C 180,E1 -14238.163,E2 -14238.163} C_VEL
LIN {X 0,Y 346.076,Z 441.498,A -85,B 0,C 180,E1 -14239.368,E2 -14239.368} C_VEL
LIN {X 0,Y 346.311,Z 423.949,A -85,B 0,C 180,E1 -14239.865,E2 -14239.865} C_VEL
LIN {X 0,Y 341.027,Z 407.191,A -85,B 0,C 180,E1 -14240.578,E2 -14240.578} C_VEL
LIN {X 0,Y 340.807,Z 406.149,A -85,B 0,C 180,E1 -14240.798,E2 -14240.798} C_VEL
LIN {X 0,Y 340.748,Z 406.042,A -85,B 0,C 180,E1 -14244.836,E2 -14244.836} C_VEL
LIN {X 0,Y 340.687,Z 406.032,A -85,B 0,C 180,E1 -14248.325,E2 -14248.325} C_VEL
LIN {X 0,Y 340.696,Z 406.049,A -85,B 0,C 180,E1 -14251.045,E2 -14251.045} C_VEL
LIN {X 0,Y 340.72,Z 406.04,A -85,B 0,C 180,E1 -14255.279,E2 -14255.279} C_VEL
LIN {X 0,Y 340.711,Z 406.034,A -85,B 0,C 180,E1 -14258.386,E2 -14258.386} C_VEL
LIN {X 0,Y 340.7,Z 406.037,A -85,B 0,C 180,E1 -14262.045,E2 -14262.045} C_VEL
LIN {X 0,Y 340.653,Z 406.05,A -85,B 0,C 180,E1 -14266.227,E2 -14266.227} C_VEL
LIN {X 0,Y 340.678,Z 406.045,A -85,B 0,C 180,E1 -14269.755,E2 -14269.755} C_VEL
LIN {X 0,Y 340.765,Z 406.219,A -85,B 0,C 180,E1 -14272.57,E2 -14272.57} C_VEL
LIN {X 0,Y 345.072,Z 420.648,A -85,B 0,C 180,E1 -14275.573,E2 -14275.573} C_VEL
LIN {X 0,Y 348.363,Z 433.885,A -85,B 0,C 180,E1 -14278.147,E2 -14278.147} C_VEL
LIN {X 0,Y 349.877,Z 441.233,A -85,B 0,C 180,E1 -14279.523,E2 -14279.523} C_VEL
LIN {X 0,Y 348.69,Z 457.029,A -85,B 0,C 180,E1 -14282.056,E2 -14282.056} C_VEL
LIN {X 0,Y 347.018,Z 479.906,A -85,B 0,C 180,E1 -14285.569,E2 -14285.569} C_VEL
LIN {X 0,Y 346.517,Z 488.117,A -85,B 0,C 180,E1 -14286.749,E2 -14286.749} C_VEL
LIN {X 0,Y 350.567,Z 516.204,A -85,B 0,C 180,E1 -14287.653,E2 -14287.653} C_VEL
LIN {X 0,Y 349.032,Z 598.653,A -85,B 0,C 180,E1 -14289.367,E2 -14289.367} C_VEL
LIN {X 0,Y 348.362,Z 611.738,A -85,B 0,C 180,E1 -14289.827,E2 -14289.827} C_VEL
LIN {X 0,Y 347.699,Z 623.154,A -85,B 0,C 180,E1 -14290.441,E2 -14290.441} C_VEL
LIN {X 0,Y 346.543,Z 635.859,A -85,B 0,C 180,E1 -14291.373,E2 -14291.373} C_VEL
LIN {X 0,Y 345.301,Z 647.832,A -85,B 0,C 180,E1 -14292.53,E2 -14292.53} C_VEL
LIN {X 0,Y 344.135,Z 658.262,A -85,B 0,C 180,E1 -14293.826,E2 -14293.826} C_VEL
LIN {X 0,Y 343.145,Z 667.025,A -85,B 0,C 180,E1 -14295.166,E2 -14295.166} C_VEL
LIN {X 0,Y 341.815,Z 676.429,A -85,B 0,C 180,E1 -14296.928,E2 -14296.928} C_VEL
LIN {X 0,Y 340.901,Z 683.899,A -85,B 0,C 180,E1 -14298.706,E2 -14298.706} C_VEL
LIN {X 0,Y 340.175,Z 689.895,A -85,B 0,C 180,E1 -14300.487,E2 -14300.487} C_VEL
LIN {X 0,Y 339.681,Z 694.638,A -85,B 0,C 180,E1 -14302.271,E2 -14302.271} C_VEL
LIN {X 0,Y 339.347,Z 698.269,A -85,B 0,C 180,E1 -14304.056,E2 -14304.056} C_VEL
LIN {X 0,Y 339.209,Z 700.138,A -85,B 0,C 180,E1 -14305.246,E2 -14305.246} C_VEL
LIN {X 0,Y 339.1,Z 701.566,A -85,B 0,C 180,E1 -14306.435,E2 -14306.435} C_VEL
LIN {X 0,Y 338.967,Z 703.184,A -85,B 0,C 180,E1 -14308.812,E2 -14308.812} C_VEL
LIN {X 0,Y 338.979,Z 703.419,A -85,B 0,C 180,E1 -14310,E2 -14310} C_VEL
LIN {X 0,Y 338.967,Z 703.224,A -85,B 0,C 180,E1 -14311.188,E2 -14311.188} C_VEL
LIN {X 0,Y 339.098,Z 701.661,A -85,B 0,C 180,E1 -14313.565,E2 -14313.565} C_VEL
LIN {X 0,Y 339.2,Z 700.286,A -85,B 0,C 180,E1 -14314.754,E2 -14314.754} C_VEL
LIN {X 0,Y 339.338,Z 697.98,A -85,B 0,C 180,E1 -14316.212,E2 -14316.212} C_VEL
LIN {X 0,Y 339.75,Z 693.475,A -85,B 0,C 180,E1 -14318.326,E2 -14318.326} C_VEL
LIN {X 0,Y 340.329,Z 688.392,A -85,B 0,C 180,E1 -14320.11,E2 -14320.11} C_VEL
LIN {X 0,Y 341.116,Z 681.986,A -85,B 0,C 180,E1 -14321.89,E2 -14321.89} C_VEL
LIN {X 0,Y 342.221,Z 674.027,A -85,B 0,C 180,E1 -14323.661,E2 -14323.661} C_VEL
LIN {X 0,Y 343.308,Z 665.895,A -85,B 0,C 180,E1 -14325.13,E2 -14325.13} C_VEL
LIN {X 0,Y 344.416,Z 655.894,A -85,B 0,C 180,E1 -14326.6,E2 -14326.6} C_VEL
LIN {X 0,Y 345.509,Z 646.029,A -85,B 0,C 180,E1 -14327.765,E2 -14327.765} C_VEL
LIN {X 0,Y 346.662,Z 635.329,A -85,B 0,C 180,E1 -14328.774,E2 -14328.774} C_VEL
LIN {X 0,Y 347.39,Z 626.736,A -85,B 0,C 180,E1 -14329.428,E2 -14329.428} C_VEL
LIN {X 0,Y 347.248,Z 621.287,A -85,B 0,C 180,E1 -14329.812,E2 -14329.812} C_VEL
LIN {X 0,Y 345.08,Z 612.38,A -85,B 0,C 180,E1 -14330.451,E2 -14330.451} C_VEL
LIN {X 0,Y 342.845,Z 603.279,A -85,B 0,C 180,E1 -14330.98,E2 -14330.98} C_VEL
LIN {X 0,Y 342.512,Z 597.536,A -85,B 0,C 180,E1 -14331.184,E2 -14331.184} C_VEL
LIN {X 0,Y 343.965,Z 516.356,A -85,B 0,C 180,E1 -14332.903,E2 -14332.903} C_VEL
LIN {X 0,Y 339.904,Z 487.829,A -85,B 0,C 180,E1 -14333.86,E2 -14333.86} C_VEL
LIN {X 0,Y 341.026,Z 470.588,A -85,B 0,C 180,E1 -14336.466,E2 -14336.466} C_VEL
LIN {X 0,Y 342.955,Z 447.848,A -85,B 0,C 180,E1 -14340.077,E2 -14340.077} C_VEL
LIN {X 0,Y 343.292,Z 443.548,A -85,B 0,C 180,E1 -14340.785,E2 -14340.785} C_VEL
LIN {X 0,Y 340.934,Z 432.555,A -85,B 0,C 180,E1 -14342.896,E2 -14342.896} C_VEL
LIN {X 0,Y 337.318,Z 418.826,A -85,B 0,C 180,E1 -14345.652,E2 -14345.652} C_VEL
LIN {X 0,Y 333.709,Z 407.133,A -85,B 0,C 180,E1 -14348.168,E2 -14348.168} C_VEL
LIN {X 0,Y 333.64,Z 406.928,A -85,B 0,C 180,E1 -14352.382,E2 -14352.382} C_VEL
LIN {X 0,Y 333.597,Z 406.912,A -85,B 0,C 180,E1 -14355.955,E2 -14355.955} C_VEL
LIN {X 0,Y 333.605,Z 406.925,A -85,B 0,C 180,E1 -14359.325,E2 -14359.325} C_VEL
LIN {X 0,Y 333.664,Z 406.913,A -85,B 0,C 180,E1 -14363.169,E2 -14363.169} C_VEL
LIN {X 0,Y 333.675,Z 406.918,A -85,B 0,C 180,E1 -14365.341,E2 -14365.341} C_VEL
LIN {X 0,Y 333.633,Z 406.928,A -85,B 0,C 180,E1 -14368.222,E2 -14368.222} C_VEL
LIN {X 0,Y 333.634,Z 406.914,A -85,B 0,C 180,E1 -14371.02,E2 -14371.02} C_VEL
LIN {X 0,Y 333.698,Z 406.913,A -85,B 0,C 180,E1 -14375.088,E2 -14375.088} C_VEL
LIN {X 0,Y 333.659,Z 406.923,A -85,B 0,C 180,E1 -14379.018,E2 -14379.018} C_VEL
LIN {X 0,Y 333.717,Z 406.899,A -85,B 0,C 180,E1 -14381.585,E2 -14381.585} C_VEL
LIN {X 0,Y 333.777,Z 406.911,A -85,B 0,C 180,E1 -14385.6,E2 -14385.6} C_VEL
LIN {X 0,Y 333.817,Z 406.88,A -85,B 0,C 180,E1 -14389.077,E2 -14389.077} C_VEL
LIN {X 0,Y 333.959,Z 406.882,A -85,B 0,C 180,E1 -14392.746,E2 -14392.746} C_VEL
LIN {X 0,Y 333.777,Z 406.885,A -85,B 0,C 180,E1 -14395.169,E2 -14395.169} C_VEL
LIN {X 0,Y 334.067,Z 406.864,A -85,B 0,C 180,E1 -14397.588,E2 -14397.588} C_VEL
LIN {X 0,Y 334.061,Z 406.858,A -85,B 0,C 180,E1 -14401.205,E2 -14401.205} C_VEL
LIN {X 0,Y 334.062,Z 406.847,A -85,B 0,C 180,E1 -14402.411,E2 -14402.411} C_VEL
LIN {X 0,Y 333.992,Z 406.883,A -85,B 0,C 180,E1 -14406.039,E2 -14406.039} C_VEL
LIN {X 0,Y 333.916,Z 406.875,A -85,B 0,C 180,E1 -14408.472,E2 -14408.472} C_VEL
LIN {X 0,Y 333.789,Z 406.905,A -85,B 0,C 180,E1 -14412.155,E2 -14412.155} C_VEL
LIN {X 0,Y 333.736,Z 406.906,A -85,B 0,C 180,E1 -14414.638,E2 -14414.638} C_VEL
LIN {X 0,Y 333.692,Z 406.915,A -85,B 0,C 180,E1 -14418.6,E2 -14418.6} C_VEL
LIN {X 0,Y 333.651,Z 406.906,A -85,B 0,C 180,E1 -14422.281,E2 -14422.281} C_VEL
LIN {X 0,Y 333.661,Z 406.918,A -85,B 0,C 180,E1 -14425.078,E2 -14425.078} C_VEL
LIN {X 0,Y 333.633,Z 406.907,A -85,B 0,C 180,E1 -14428.98,E2 -14428.98} C_VEL
LIN {X 0,Y 333.646,Z 406.922,A -85,B 0,C 180,E1 -14432.587,E2 -14432.587} C_VEL
LIN {X 0,Y 333.675,Z 406.919,A -85,B 0,C 180,E1 -14436.139,E2 -14436.139} C_VEL
LIN {X 0,Y 333.603,Z 406.905,A -85,B 0,C 180,E1 -14439.199,E2 -14439.199} C_VEL
LIN {X 0,Y 333.627,Z 406.882,A -85,B 0,C 180,E1 -14442.498,E2 -14442.498} C_VEL
LIN {X 0,Y 333.595,Z 406.929,A -85,B 0,C 180,E1 -14445.954,E2 -14445.954} C_VEL
LIN {X 0,Y 333.603,Z 406.89,A -85,B 0,C 180,E1 -14449.325,E2 -14449.325} C_VEL
LIN {X 0,Y 333.662,Z 406.924,A -85,B 0,C 180,E1 -14453.169,E2 -14453.169} C_VEL
LIN {X 0,Y 333.758,Z 407.212,A -85,B 0,C 180,E1 -14454.47,E2 -14454.47} C_VEL
LIN {X 0,Y 337.599,Z 424.931,A -85,B 0,C 180,E1 -14458.289,E2 -14458.289} C_VEL
LIN {X 0,Y 339.476,Z 434.188,A -85,B 0,C 180,E1 -14460.207,E2 -14460.207} C_VEL
LIN {X 0,Y 337.823,Z 450.177,A -85,B 0,C 180,E1 -14463.247,E2 -14463.247} C_VEL
LIN {X 0,Y 337.472,Z 453.872,A -85,B 0,C 180,E1 -14463.92,E2 -14463.92} C_VEL
LIN {X 0,Y 339.43,Z 486.393,A -85,B 0,C 180,E1 -14466.186,E2 -14466.186} C_VEL
LIN {X 0,Y 339.587,Z 489.14,A -85,B 0,C 180,E1 -14466.347,E2 -14466.347} C_VEL
LIN {X 0,Y 342.63,Z 516.176,A -85,B 0,C 180,E1 -14467.172,E2 -14467.172} C_VEL
LIN {X 0,Y 343.419,Z 525.304,A -85,B 0,C 180,E1 -14467.429,E2 -14467.429} C_VEL
LIN {X 0,Y 341.872,Z 605.304,A -85,B 0,C 180,E1 -14469.112,E2 -14469.112} C_VEL
LIN {X 0,Y 341.175,Z 618.111,A -85,B 0,C 180,E1 -14469.58,E2 -14469.58} C_VEL
LIN {X 0,Y 340.283,Z 631.018,A -85,B 0,C 180,E1 -14470.311,E2 -14470.311} C_VEL
LIN {X 0,Y 339.165,Z 643.291,A -85,B 0,C 180,E1 -14471.265,E2 -14471.265} C_VEL
LIN {X 0,Y 337.868,Z 654.798,A -85,B 0,C 180,E1 -14472.445,E2 -14472.445} C_VEL
LIN {X 0,Y 336.668,Z 665.183,A -85,B 0,C 180,E1 -14473.793,E2 -14473.793} C_VEL
LIN {X 0,Y 335.675,Z 673.586,A -85,B 0,C 180,E1 -14475.139,E2 -14475.139} C_VEL
LIN {X 0,Y 334.443,Z 682.699,A -85,B 0,C 180,E1 -14476.944,E2 -14476.944} C_VEL
LIN {X 0,Y 333.541,Z 690.013,A -85,B 0,C 180,E1 -14478.761,E2 -14478.761} C_VEL
LIN {X 0,Y 332.763,Z 696.705,A -85,B 0,C 180,E1 -14480.886,E2 -14480.886} C_VEL
LIN {X 0,Y 332.344,Z 701.094,A -85,B 0,C 180,E1 -14482.71,E2 -14482.71} C_VEL
LIN {X 0,Y 332.181,Z 703.404,A -85,B 0,C 180,E1 -14483.927,E2 -14483.927} C_VEL
LIN {X 0,Y 332.105,Z 705.286,A -85,B 0,C 180,E1 -14485.144,E2 -14485.144} C_VEL
LIN {X 0,Y 332.06,Z 706.704,A -85,B 0,C 180,E1 -14486.359,E2 -14486.359} C_VEL
LIN {X 0,Y 331.946,Z 708.316,A -85,B 0,C 180,E1 -14488.787,E2 -14488.787} C_VEL
LIN {X 0,Y 331.982,Z 708.533,A -85,B 0,C 180,E1 -14490,E2 -14490} C_VEL
LIN {X 0,Y 331.985,Z 708.311,A -85,B 0,C 180,E1 -14491.213,E2 -14491.213} C_VEL
LIN {X 0,Y 332.066,Z 706.692,A -85,B 0,C 180,E1 -14493.64,E2 -14493.64} C_VEL
LIN {X 0,Y 332.115,Z 705.266,A -85,B 0,C 180,E1 -14494.855,E2 -14494.855} C_VEL
LIN {X 0,Y 332.256,Z 702.302,A -85,B 0,C 180,E1 -14496.68,E2 -14496.68} C_VEL
LIN {X 0,Y 332.589,Z 698.273,A -85,B 0,C 180,E1 -14498.506,E2 -14498.506} C_VEL
LIN {X 0,Y 333.27,Z 692.059,A -85,B 0,C 180,E1 -14500.633,E2 -14500.633} C_VEL
LIN {X 0,Y 334.113,Z 685.276,A -85,B 0,C 180,E1 -14502.451,E2 -14502.451} C_VEL
LIN {X 0,Y 335.023,Z 678.331,A -85,B 0,C 180,E1 -14503.96,E2 -14503.96} C_VEL
LIN {X 0,Y 336.067,Z 669.935,A -85,B 0,C 180,E1 -14505.464,E2 -14505.464} C_VEL
LIN {X 0,Y 337.302,Z 659.539,A -85,B 0,C 180,E1 -14506.96,E2 -14506.96} C_VEL
LIN {X 0,Y 338.48,Z 649.236,A -85,B 0,C 180,E1 -14508.147,E2 -14508.147} C_VEL
LIN {X 0,Y 339.674,Z 637.888,A -85,B 0,C 180,E1 -14509.175,E2 -14509.175} C_VEL
LIN {X 0,Y 340.607,Z 626.123,A -85,B 0,C 180,E1 -14509.983,E2 -14509.983} C_VEL
LIN {X 0,Y 341.462,Z 613.468,A -85,B 0,C 180,E1 -14510.599,E2 -14510.599} C_VEL
LIN {X 0,Y 341.714,Z 609.173,A -85,B 0,C 180,E1 -14510.78,E2 -14510.78} C_VEL
LIN {X 0,Y 343.923,Z 594.879,A -85,B 0,C 180,E1 -14511.818,E2 -14511.818} C_VEL
LIN {X 0,Y 345.616,Z 580.314,A -85,B 0,C 180,E1 -14512.61,E2 -14512.61} C_VEL
LIN {X 0,Y 346.863,Z 564.878,A -85,B 0,C 180,E1 -14513.193,E2 -14513.193} C_VEL
LIN {X 0,Y 349.234,Z 524.735,A -85,B 0,C 180,E1 -14514.515,E2 -14514.515} C_VEL
LIN {X 0,Y 348.615,Z 505.003,A -85,B 0,C 180,E1 -14515.437,E2 -14515.437} C_VEL
LIN {X 0,Y 347.021,Z 487.798,A -85,B 0,C 180,E1 -14516.437,E2 -14516.437} C_VEL
LIN {X 0,Y 344.652,Z 471.547,A -85,B 0,C 180,E1 -14517.577,E2 -14517.577} C_VEL
LIN {X 0,Y 342.379,Z 458.813,A -85,B 0,C 180,E1 -14518.625,E2 -14518.625} C_VEL
LIN {X 0,Y 341.665,Z 454.461,A -85,B 0,C 180,E1 -14519.033,E2 -14519.033} C_VEL
LIN {X 0,Y 343.752,Z 443.899,A -85,B 0,C 180,E1 -14521.423,E2 -14521.423} C_VEL
LIN {X 0,Y 342.528,Z 436.54,A -85,B 0,C 180,E1 -14523.641,E2 -14523.641} C_VEL
LIN {X 0,Y 340.635,Z 428.705,A -85,B 0,C 180,E1 -14526.423,E2 -14526.423} C_VEL
LIN {X 0,Y 338.974,Z 422.975,A -85,B 0,C 180,E1 -14528.842,E2 -14528.842} C_VEL
LIN {X 0,Y 337.392,Z 417.947,A -85,B 0,C 180,E1 -14531.419,E2 -14531.419} C_VEL
LIN {X 0,Y 336.162,Z 414.494,A -85,B 0,C 180,E1 -14533.624,E2 -14533.624} C_VEL
LIN {X 0,Y 335.054,Z 411.358,A -85,B 0,C 180,E1 -14536.196,E2 -14536.196} C_VEL
LIN {X 0,Y 334.642,Z 409.814,A -85,B 0,C 180,E1 -14537.774,E2 -14537.774} C_VEL
LIN {X 0,Y 333.796,Z 407.826,A -85,B 0,C 180,E1 -14541.172,E2 -14541.172} C_VEL
LIN {X 0,Y 333.701,Z 407.181,A -85,B 0,C 180,E1 -14543.864,E2 -14543.864} C_VEL
LIN {X 0,Y 333.741,Z 407.498,A -85,B 0,C 180,E1 -14546.803,E2 -14546.803} C_VEL
LIN {X 0,Y 334.137,Z 408.768,A -85,B 0,C 180,E1 -14549.352,E2 -14549.352} C_VEL
LIN {X 0,Y 336.103,Z 411.441,A -85,B 0,C 180,E1 -14550.144,E2 -14550.144} C_VEL
LIN {X 0,Y 337.302,Z 412.644,A -85,B 0,C 180,E1 -14550.533,E2 -14550.533} C_VEL
LIN {X 0,Y 339.303,Z 415.944,A -85,B 0,C 180,E1 -14551.221,E2 -14551.221} C_VEL
LIN {X 0,Y 340.587,Z 417.55,A -85,B 0,C 180,E1 -14551.604,E2 -14551.604} C_VEL
LIN {X 0,Y 342.944,Z 421.059,A -85,B 0,C 180,E1 -14552.319,E2 -14552.319} C_VEL
LIN {X 0,Y 347.77,Z 428.976,A -85,B 0,C 180,E1 -14553.677,E2 -14553.677} C_VEL
LIN {X 0,Y 352.728,Z 438.256,A -85,B 0,C 180,E1 -14554.969,E2 -14554.969} C_VEL
LIN {X 0,Y 353.679,Z 440.32,A -85,B 0,C 180,E1 -14555.223,E2 -14555.223} C_VEL
LIN {X 0,Y 350.36,Z 486.425,A -85,B 0,C 180,E1 -14556.817,E2 -14556.817} C_VEL
LIN {X 0,Y 349.626,Z 504.256,A -85,B 0,C 180,E1 -14557.547,E2 -14557.547} C_VEL
LIN {X 0,Y 348.992,Z 516.514,A -85,B 0,C 180,E1 -14558.248,E2 -14558.248} C_VEL
LIN {X 0,Y 347.943,Z 528.708,A -85,B 0,C 180,E1 -14559.171,E2 -14559.171} C_VEL
LIN {X 0,Y 346.668,Z 540.361,A -85,B 0,C 180,E1 -14560.303,E2 -14560.303} C_VEL
LIN {X 0,Y 345.099,Z 550.97,A -85,B 0,C 180,E1 -14561.599,E2 -14561.599} C_VEL
LIN {X 0,Y 343.607,Z 560.602,A -85,B 0,C 180,E1 -14563.054,E2 -14563.054} C_VEL
LIN {X 0,Y 342.215,Z 568.421,A -85,B 0,C 180,E1 -14564.515,E2 -14564.515} C_VEL
LIN {X 0,Y 340.447,Z 576.525,A -85,B 0,C 180,E1 -14566.398,E2 -14566.398} C_VEL
LIN {X 0,Y 339.153,Z 582.094,A -85,B 0,C 180,E1 -14568.04,E2 -14568.04} C_VEL
LIN {X 0,Y 337.936,Z 586.855,A -85,B 0,C 180,E1 -14569.818,E2 -14569.818} C_VEL
LIN {X 0,Y 336.821,Z 590.43,A -85,B 0,C 180,E1 -14571.601,E2 -14571.601} C_VEL
LIN {X 0,Y 336.162,Z 592.182,A -85,B 0,C 180,E1 -14572.794,E2 -14572.794} C_VEL
LIN {X 0,Y 335.664,Z 593.479,A -85,B 0,C 180,E1 -14573.991,E2 -14573.991} C_VEL
LIN {X 0,Y 335.345,Z 594.331,A -85,B 0,C 180,E1 -14575.191,E2 -14575.191} C_VEL
LIN {X 0,Y 334.963,Z 594.745,A -85,B 0,C 180,E1 -14576.391,E2 -14576.391} C_VEL
LIN {X 0,Y 334.626,Z 594.742,A -85,B 0,C 180,E1 -14577.593,E2 -14577.593} C_VEL
LIN {X 0,Y 334.309,Z 594.329,A -85,B 0,C 180,E1 -14578.795,E2 -14578.795} C_VEL
LIN {X 0,Y 333.979,Z 593.465,A -85,B 0,C 180,E1 -14580,E2 -14580} C_VEL
LIN {X 0,Y 333.984,Z 592.128,A -85,B 0,C 180,E1 -14581.206,E2 -14581.206} C_VEL
LIN {X 0,Y 333.89,Z 589.323,A -85,B 0,C 180,E1 -14583.016,E2 -14583.016} C_VEL
LIN {X 0,Y 333.828,Z 585.466,A -85,B 0,C 180,E1 -14584.831,E2 -14584.831} C_VEL
LIN {X 0,Y 334.195,Z 580.43,A -85,B 0,C 180,E1 -14586.642,E2 -14586.642} C_VEL
LIN {X 0,Y 334.546,Z 574.111,A -85,B 0,C 180,E1 -14588.456,E2 -14588.456} C_VEL
LIN {X 0,Y 334.948,Z 566.19,A -85,B 0,C 180,E1 -14590.274,E2 -14590.274} C_VEL
LIN {X 0,Y 335.535,Z 556.393,A -85,B 0,C 180,E1 -14592.091,E2 -14592.091} C_VEL
LIN {X 0,Y 336.039,Z 546.242,A -85,B 0,C 180,E1 -14593.609,E2 -14593.609} C_VEL
LIN {X 0,Y 336.627,Z 535.042,A -85,B 0,C 180,E1 -14594.973,E2 -14594.973} C_VEL
LIN {X 0,Y 337.278,Z 522.667,A -85,B 0,C 180,E1 -14596.17,E2 -14596.17} C_VEL
LIN {X 0,Y 337.7,Z 509.385,A -85,B 0,C 180,E1 -14597.173,E2 -14597.173} C_VEL
LIN {X 0,Y 338.066,Z 495.456,A -85,B 0,C 180,E1 -14597.935,E2 -14597.935} C_VEL
LIN {X 0,Y 338.304,Z 482.105,A -85,B 0,C 180,E1 -14598.431,E2 -14598.431} C_VEL
LIN {X 0,Y 339.066,Z 442.43,A -85,B 0,C 180,E1 -14599.569,E2 -14599.569} C_VEL
LIN {X 0,Y 339.446,Z 425.433,A -85,B 0,C 180,E1 -14600.069,E2 -14600.069} C_VEL
LIN {X 0,Y 333.906,Z 407.752,A -85,B 0,C 180,E1 -14600.848,E2 -14600.848} C_VEL
LIN {X 0,Y 333.762,Z 406.969,A -85,B 0,C 180,E1 -14601.089,E2 -14601.089} C_VEL
LIN {X 0,Y 333.699,Z 406.92,A -85,B 0,C 180,E1 -14605.093,E2 -14605.093} C_VEL
LIN {X 0,Y 333.657,Z 406.906,A -85,B 0,C 180,E1 -14608.977,E2 -14608.977} C_VEL
LIN {X 0,Y 333.645,Z 406.918,A -85,B 0,C 180,E1 -14612.587,E2 -14612.587} C_VEL
LIN {X 0,Y 333.678,Z 406.921,A -85,B 0,C 180,E1 -14616.139,E2 -14616.139} C_VEL
LIN {X 0,Y 333.648,Z 406.919,A -85,B 0,C 180,E1 -14619.192,E2 -14619.192} C_VEL
LIN {X 0,Y 333.634,Z 406.919,A -85,B 0,C 180,E1 -14622.5,E2 -14622.5} C_VEL
LIN {X 0,Y 333.598,Z 406.926,A -85,B 0,C 180,E1 -14625.955,E2 -14625.955} C_VEL
LIN {X 0,Y 333.645,Z 406.927,A -85,B 0,C 180,E1 -14629.316,E2 -14629.316} C_VEL
LIN {X 0,Y 333.727,Z 407.122,A -85,B 0,C 180,E1 -14631.953,E2 -14631.953} C_VEL
LIN {X 0,Y 337.767,Z 420.302,A -85,B 0,C 180,E1 -14634.755,E2 -14634.755} C_VEL
LIN {X 0,Y 341.42,Z 434.693,A -85,B 0,C 180,E1 -14637.643,E2 -14637.643} C_VEL
LIN {X 0,Y 343.222,Z 443.451,A -85,B 0,C 180,E1 -14639.319,E2 -14639.319} C_VEL
LIN {X 0,Y 341.828,Z 460.973,A -85,B 0,C 180,E1 -14642.139,E2 -14642.139} C_VEL
LIN {X 0,Y 340.072,Z 484.436,A -85,B 0,C 180,E1 -14645.749,E2 -14645.749} C_VEL
LIN {X 0,Y 339.833,Z 487.928,A -85,B 0,C 180,E1 -14646.253,E2 -14646.253} C_VEL
LIN {X 0,Y 344.019,Z 517.139,A -85,B 0,C 180,E1 -14647.226,E2 -14647.226} C_VEL
LIN {X 0,Y 342.401,Z 598.645,A -85,B 0,C 180,E1 -14648.949,E2 -14648.949} C_VEL
LIN {X 0,Y 341.717,Z 611.758,A -85,B 0,C 180,E1 -14649.417,E2 -14649.417} C_VEL
LIN {X 0,Y 341.032,Z 623.188,A -85,B 0,C 180,E1 -14650.043,E2 -14650.043} C_VEL
LIN {X 0,Y 339.832,Z 635.9,A -85,B 0,C 180,E1 -14650.991,E2 -14650.991} C_VEL
LIN {X 0,Y 338.517,Z 647.878,A -85,B 0,C 180,E1 -14652.168,E2 -14652.168} C_VEL
LIN {X 0,Y 337.463,Z 657.227,A -85,B 0,C 180,E1 -14653.335,E2 -14653.335} C_VEL
LIN {X 0,Y 336.285,Z 667.076,A -85,B 0,C 180,E1 -14654.857,E2 -14654.857} C_VEL
LIN {X 0,Y 334.896,Z 676.482,A -85,B 0,C 180,E1 -14656.653,E2 -14656.653} C_VEL
LIN {X 0,Y 333.932,Z 683.952,A -85,B 0,C 180,E1 -14658.467,E2 -14658.467} C_VEL
LIN {X 0,Y 333.147,Z 689.949,A -85,B 0,C 180,E1 -14660.284,E2 -14660.284} C_VEL
LIN {X 0,Y 332.614,Z 694.693,A -85,B 0,C 180,E1 -14662.106,E2 -14662.106} C_VEL
LIN {X 0,Y 332.27,Z 698.323,A -85,B 0,C 180,E1 -14663.929,E2 -14663.929} C_VEL
LIN {X 0,Y 332.117,Z 700.192,A -85,B 0,C 180,E1 -14665.145,E2 -14665.145} C_VEL
LIN {X 0,Y 332.03,Z 701.62,A -85,B 0,C 180,E1 -14666.359,E2 -14666.359} C_VEL
LIN {X 0,Y 331.876,Z 703.238,A -85,B 0,C 180,E1 -14668.787,E2 -14668.787} C_VEL
LIN {X 0,Y 331.885,Z 703.473,A -85,B 0,C 180,E1 -14670,E2 -14670} C_VEL
LIN {X 0,Y 331.876,Z 703.278,A -85,B 0,C 180,E1 -14671.214,E2 -14671.214} C_VEL
LIN {X 0,Y 332.029,Z 701.714,A -85,B 0,C 180,E1 -14673.641,E2 -14673.641} C_VEL
LIN {X 0,Y 332.106,Z 700.339,A -85,B 0,C 180,E1 -14674.856,E2 -14674.856} C_VEL
LIN {X 0,Y 332.295,Z 697.561,A -85,B 0,C 180,E1 -14676.619,E2 -14676.619} C_VEL
LIN {X 0,Y 332.715,Z 693.526,A -85,B 0,C 180,E1 -14678.503,E2 -14678.503} C_VEL
LIN {X 0,Y 333.311,Z 688.442,A -85,B 0,C 180,E1 -14680.325,E2 -14680.325} C_VEL
LIN {X 0,Y 334.142,Z 682.034,A -85,B 0,C 180,E1 -14682.142,E2 -14682.142} C_VEL
LIN {X 0,Y 335.315,Z 674.074,A -85,B 0,C 180,E1 -14683.948,E2 -14683.948} C_VEL
LIN {X 0,Y 336.451,Z 665.939,A -85,B 0,C 180,E1 -14685.446,E2 -14685.446} C_VEL
LIN {X 0,Y 337.595,Z 655.934,A -85,B 0,C 180,E1 -14686.945,E2 -14686.945} C_VEL
LIN {X 0,Y 338.902,Z 644.688,A -85,B 0,C 180,E1 -14688.28,E2 -14688.28} C_VEL
LIN {X 0,Y 340.143,Z 633.651,A -85,B 0,C 180,E1 -14689.305,E2 -14689.305} C_VEL
LIN {X 0,Y 341.142,Z 621.186,A -85,B 0,C 180,E1 -14690.187,E2 -14690.187} C_VEL
LIN {X 0,Y 342.001,Z 608.158,A -85,B 0,C 180,E1 -14690.841,E2 -14690.841} C_VEL
LIN {X 0,Y 342.512,Z 597.536,A -85,B 0,C 180,E1 -14691.184,E2 -14691.184} C_VEL
LIN {X 0,Y 342.193,Z 591.747,A -85,B 0,C 180,E1 -14691.365,E2 -14691.365} C_VEL
LIN {X 0,Y 339.71,Z 582.414,A -85,B 0,C 180,E1 -14691.743,E2 -14691.743} C_VEL
LIN {X 0,Y 337.072,Z 573.066,A -85,B 0,C 180,E1 -14692.114,E2 -14692.114} C_VEL
LIN {X 0,Y 336.512,Z 567.246,A -85,B 0,C 180,E1 -14692.278,E2 -14692.278} C_VEL
LIN {X 0,Y 337.465,Z 517.476,A -85,B 0,C 180,E1 -14693.342,E2 -14693.342} C_VEL
LIN {X 0,Y 333.267,Z 487.812,A -85,B 0,C 180,E1 -14694.364,E2 -14694.364} C_VEL
LIN {X 0,Y 334.619,Z 468.398,A -85,B 0,C 180,E1 -14697.351,E2 -14697.351} C_VEL
LIN {X 0,Y 336.426,Z 448.202,A -85,B 0,C 180,E1 -14700.606,E2 -14700.606} C_VEL
LIN {X 0,Y 336.445,Z 444.2,A -85,B 0,C 180,E1 -14701.308,E2 -14701.308} C_VEL
LIN {X 0,Y 333.291,Z 430.457,A -85,B 0,C 180,E1 -14704.025,E2 -14704.025} C_VEL
LIN {X 0,Y 329.476,Z 416.733,A -85,B 0,C 180,E1 -14706.875,E2 -14706.875} C_VEL
LIN {X 0,Y 326.611,Z 408.022,A -85,B 0,C 180,E1 -14708.836,E2 -14708.836} C_VEL
LIN {X 0,Y 326.546,Z 407.794,A -85,B 0,C 180,E1 -14711.124,E2 -14711.124} C_VEL
LIN {X 0,Y 326.562,Z 407.79,A -85,B 0,C 180,E1 -14713.526,E2 -14713.526} C_VEL
LIN {X 0,Y 326.576,Z 407.806,A -85,B 0,C 180,E1 -14717.029,E2 -14717.029} C_VEL
LIN {X 0,Y 326.584,Z 407.805,A -85,B 0,C 180,E1 -14721.386,E2 -14721.386} C_VEL
LIN {X 0,Y 326.621,Z 407.8,A -85,B 0,C 180,E1 -14724.852,E2 -14724.852} C_VEL
LIN {X 0,Y 326.611,Z 407.791,A -85,B 0,C 180,E1 -14727.456,E2 -14727.456} C_VEL
LIN {X 0,Y 326.584,Z 407.796,A -85,B 0,C 180,E1 -14730.333,E2 -14730.333} C_VEL
LIN {X 0,Y 326.611,Z 407.8,A -85,B 0,C 180,E1 -14733.136,E2 -14733.136} C_VEL
LIN {X 0,Y 326.632,Z 407.783,A -85,B 0,C 180,E1 -14735.869,E2 -14735.869} C_VEL
LIN {X 0,Y 326.614,Z 407.799,A -85,B 0,C 180,E1 -14739.862,E2 -14739.862} C_VEL
LIN {X 0,Y 326.678,Z 407.783,A -85,B 0,C 180,E1 -14743.759,E2 -14743.759} C_VEL
LIN {X 0,Y 326.745,Z 407.78,A -85,B 0,C 180,E1 -14746.314,E2 -14746.314} C_VEL
LIN {X 0,Y 326.784,Z 407.766,A -85,B 0,C 180,E1 -14750.093,E2 -14750.093} C_VEL
LIN {X 0,Y 326.944,Z 407.746,A -85,B 0,C 180,E1 -14753.83,E2 -14753.83} C_VEL
LIN {X 0,Y 327.011,Z 407.743,A -85,B 0,C 180,E1 -14757.536,E2 -14757.536} C_VEL
LIN {X 0,Y 327.031,Z 407.732,A -85,B 0,C 180,E1 -14761.231,E2 -14761.231} C_VEL
LIN {X 0,Y 326.742,Z 407.765,A -85,B 0,C 180,E1 -14763.7,E2 -14763.7} C_VEL
LIN {X 0,Y 326.946,Z 407.759,A -85,B 0,C 180,E1 -14766.17,E2 -14766.17} C_VEL
LIN {X 0,Y 326.784,Z 407.755,A -85,B 0,C 180,E1 -14769.907,E2 -14769.907} C_VEL
LIN {X 0,Y 326.735,Z 407.786,A -85,B 0,C 180,E1 -14773.686,E2 -14773.686} C_VEL
LIN {X 0,Y 326.62,Z 407.78,A -85,B 0,C 180,E1 -14777.532,E2 -14777.532} C_VEL
LIN {X 0,Y 326.609,Z 407.792,A -85,B 0,C 180,E1 -14781.457,E2 -14781.457} C_VEL
LIN {X 0,Y 326.603,Z 407.799,A -85,B 0,C 180,E1 -14785.491,E2 -14785.491} C_VEL
LIN {X 0,Y 326.593,Z 407.787,A -85,B 0,C 180,E1 -14788.257,E2 -14788.257} C_VEL
LIN {X 0,Y 326.576,Z 407.802,A -85,B 0,C 180,E1 -14791.097,E2 -14791.097} C_VEL
LIN {X 0,Y 326.609,Z 407.787,A -85,B 0,C 180,E1 -14794.019,E2 -14794.019} C_VEL
LIN {X 0,Y 326.624,Z 407.8,A -85,B 0,C 180,E1 -14797.237,E2 -14797.237} C_VEL
LIN {X 0,Y 326.544,Z 407.756,A -85,B 0,C 180,E1 -14801.124,E2 -14801.124} C_VEL
LIN {X 0,Y 326.56,Z 407.782,A -85,B 0,C 180,E1 -14803.526,E2 -14803.526} C_VEL
LIN {X 0,Y 326.573,Z 407.786,A -85,B 0,C 180,E1 -14807.029,E2 -14807.029} C_VEL
LIN {X 0,Y 326.583,Z 407.801,A -85,B 0,C 180,E1 -14811.385,E2 -14811.385} C_VEL
LIN {X 0,Y 326.697,Z 408.014,A -85,B 0,C 180,E1 -14814.182,E2 -14814.182} C_VEL
LIN {X 0,Y 330.246,Z 424.63,A -85,B 0,C 180,E1 -14817.857,E2 -14817.857} C_VEL
LIN {X 0,Y 332.474,Z 435.105,A -85,B 0,C 180,E1 -14820.075,E2 -14820.075} C_VEL
LIN {X 0,Y 330.788,Z 450.781,A -85,B 0,C 180,E1 -14823.109,E2 -14823.109} C_VEL
LIN {X 0,Y 331.418,Z 460.08,A -85,B 0,C 180,E1 -14823.81,E2 -14823.81} C_VEL
LIN {X 0,Y 333.029,Z 489.372,A -85,B 0,C 180,E1 -14825.855,E2 -14825.855} C_VEL
LIN {X 0,Y 336.198,Z 517.839,A -85,B 0,C 180,E1 -14826.745,E2 -14826.745} C_VEL
LIN {X 0,Y 336.875,Z 525.709,A -85,B 0,C 180,E1 -14826.973,E2 -14826.973} C_VEL
LIN {X 0,Y 335.242,Z 605.353,A -85,B 0,C 180,E1 -14828.679,E2 -14828.679} C_VEL
LIN {X 0,Y 334.541,Z 618.106,A -85,B 0,C 180,E1 -14829.156,E2 -14829.156} C_VEL
LIN {X 0,Y 333.605,Z 630.997,A -85,B 0,C 180,E1 -14829.9,E2 -14829.9} C_VEL
LIN {X 0,Y 332.449,Z 643.259,A -85,B 0,C 180,E1 -14830.872,E2 -14830.872} C_VEL
LIN {X 0,Y 331.092,Z 654.759,A -85,B 0,C 180,E1 -14832.074,E2 -14832.074} C_VEL
LIN {X 0,Y 329.752,Z 665.867,A -85,B 0,C 180,E1 -14833.554,E2 -14833.554} C_VEL
LIN {X 0,Y 328.544,Z 675.189,A -85,B 0,C 180,E1 -14835.126,E2 -14835.126} C_VEL
LIN {X 0,Y 327.302,Z 683.996,A -85,B 0,C 180,E1 -14836.97,E2 -14836.97} C_VEL
LIN {X 0,Y 326.407,Z 691.049,A -85,B 0,C 180,E1 -14838.826,E2 -14838.826} C_VEL
LIN {X 0,Y 325.749,Z 696.653,A -85,B 0,C 180,E1 -14840.688,E2 -14840.688} C_VEL
LIN {X 0,Y 325.286,Z 701.041,A -85,B 0,C 180,E1 -14842.551,E2 -14842.551} C_VEL
LIN {X 0,Y 325.082,Z 703.667,A -85,B 0,C 180,E1 -14843.98,E2 -14843.98} C_VEL
LIN {X 0,Y 324.966,Z 706.651,A -85,B 0,C 180,E1 -14846.28,E2 -14846.28} C_VEL
LIN {X 0,Y 324.893,Z 707.651,A -85,B 0,C 180,E1 -14847.52,E2 -14847.52} C_VEL
LIN {X 0,Y 324.855,Z 708.262,A -85,B 0,C 180,E1 -14848.76,E2 -14848.76} C_VEL
LIN {X 0,Y 324.887,Z 708.479,A -85,B 0,C 180,E1 -14850,E2 -14850} C_VEL
LIN {X 0,Y 324.891,Z 708.256,A -85,B 0,C 180,E1 -14851.239,E2 -14851.239} C_VEL
LIN {X 0,Y 324.994,Z 706.638,A -85,B 0,C 180,E1 -14853.72,E2 -14853.72} C_VEL
LIN {X 0,Y 325.098,Z 703.596,A -85,B 0,C 180,E1 -14856.046,E2 -14856.046} C_VEL
LIN {X 0,Y 325.404,Z 699.663,A -85,B 0,C 180,E1 -14858.07,E2 -14858.07} C_VEL
LIN {X 0,Y 325.94,Z 694.869,A -85,B 0,C 180,E1 -14859.933,E2 -14859.933} C_VEL
LIN {X 0,Y 326.671,Z 688.8,A -85,B 0,C 180,E1 -14861.793,E2 -14861.793} C_VEL
LIN {X 0,Y 327.715,Z 681.229,A -85,B 0,C 180,E1 -14863.645,E2 -14863.645} C_VEL
LIN {X 0,Y 328.788,Z 673.44,A -85,B 0,C 180,E1 -14865.18,E2 -14865.18} C_VEL
LIN {X 0,Y 329.981,Z 663.863,A -85,B 0,C 180,E1 -14866.718,E2 -14866.718} C_VEL
LIN {X 0,Y 331.278,Z 653.339,A -85,B 0,C 180,E1 -14868.075,E2 -14868.075} C_VEL
LIN {X 0,Y 332.415,Z 643.081,A -85,B 0,C 180,E1 -14869.129,E2 -14869.129} C_VEL
LIN {X 0,Y 333.573,Z 630.745,A -85,B 0,C 180,E1 -14870.102,E2 -14870.102} C_VEL
LIN {X 0,Y 334.525,Z 617.771,A -85,B 0,C 180,E1 -14870.845,E2 -14870.845} C_VEL
LIN {X 0,Y 335.021,Z 611.382,A -85,B 0,C 180,E1 -14871.134,E2 -14871.134} C_VEL
LIN {X 0,Y 337.28,Z 598.24,A -85,B 0,C 180,E1 -14872.19,E2 -14872.19} C_VEL
LIN {X 0,Y 339.153,Z 584.745,A -85,B 0,C 180,E1 -14873.025,E2 -14873.025} C_VEL
LIN {X 0,Y 340.605,Z 571.198,A -85,B 0,C 180,E1 -14873.645,E2 -14873.645} C_VEL
LIN {X 0,Y 343.573,Z 525.585,A -85,B 0,C 180,E1 -14875.216,E2 -14875.216} C_VEL
LIN {X 0,Y 343.163,Z 506.997,A -85,B 0,C 180,E1 -14876.112,E2 -14876.112} C_VEL
LIN {X 0,Y 341.708,Z 489.51,A -85,B 0,C 180,E1 -14877.169,E2 -14877.169} C_VEL
LIN {X 0,Y 339.498,Z 473.172,A -85,B 0,C 180,E1 -14878.377,E2 -14878.377} C_VEL
LIN {X 0,Y 336.827,Z 457.567,A -85,B 0,C 180,E1 -14879.74,E2 -14879.74} C_VEL
LIN {X 0,Y 335.95,Z 452.193,A -85,B 0,C 180,E1 -14880.292,E2 -14880.292} C_VEL
LIN {X 0,Y 337.194,Z 446.008,A -85,B 0,C 180,E1 -14881.754,E2 -14881.754} C_VEL
LIN {X 0,Y 335.739,Z 437.686,A -85,B 0,C 180,E1 -14884.415,E2 -14884.415} C_VEL
LIN {X 0,Y 334.107,Z 430.962,A -85,B 0,C 180,E1 -14886.933,E2 -14886.933} C_VEL
LIN {X 0,Y 332.331,Z 424.692,A -85,B 0,C 180,E1 -14889.781,E2 -14889.781} C_VEL
LIN {X 0,Y 330.545,Z 419.358,A -85,B 0,C 180,E1 -14892.873,E2 -14892.873} C_VEL
LIN {X 0,Y 329.424,Z 416.193,A -85,B 0,C 180,E1 -14895.249,E2 -14895.249} C_VEL
LIN {X 0,Y 328.361,Z 413.097,A -85,B 0,C 180,E1 -14898.514,E2 -14898.514} C_VEL
LIN {X 0,Y 327.75,Z 411.485,A -85,B 0,C 180,E1 -14901.548,E2 -14901.548} C_VEL
LIN {X 0,Y 327.708,Z 411.019,A -85,B 0,C 180,E1 -14903.095,E2 -14903.095} C_VEL
LIN {X 0,Y 327.639,Z 411.055,A -85,B 0,C 180,E1 -14906.102,E2 -14906.102} C_VEL
LIN {X 0,Y 327.872,Z 411.721,A -85,B 0,C 180,E1 -14907.714,E2 -14907.714} C_VEL
LIN {X 0,Y 330.431,Z 414.476,A -85,B 0,C 180,E1 -14908.831,E2 -14908.831} C_VEL
LIN {X 0,Y 331.539,Z 415.693,A -85,B 0,C 180,E1 -14909.232,E2 -14909.232} C_VEL
LIN {X 0,Y 334.066,Z 418.667,A -85,B 0,C 180,E1 -14910.134,E2 -14910.134} C_VEL
LIN {X 0,Y 336.278,Z 422.094,A -85,B 0,C 180,E1 -14910.919,E2 -14910.919} C_VEL
LIN {X 0,Y 340.419,Z 428.507,A -85,B 0,C 180,E1 -14912.236,E2 -14912.236} C_VEL
LIN {X 0,Y 345.529,Z 437.366,A -85,B 0,C 180,E1 -14913.72,E2 -14913.72} C_VEL
LIN {X 0,Y 348.379,Z 443.2,A -85,B 0,C 180,E1 -14914.509,E2 -14914.509} C_VEL
LIN {X 0,Y 344.87,Z 486.942,A -85,B 0,C 180,E1 -14916.079,E2 -14916.079} C_VEL
LIN {X 0,Y 344.126,Z 504.539,A -85,B 0,C 180,E1 -14916.803,E2 -14916.803} C_VEL
LIN {X 0,Y 343.335,Z 517.601,A -85,B 0,C 180,E1 -14917.561,E2 -14917.561} C_VEL
LIN {X 0,Y 342.231,Z 529.328,A -85,B 0,C 180,E1 -14918.464,E2 -14918.464} C_VEL
LIN {X 0,Y 340.832,Z 541.289,A -85,B 0,C 180,E1 -14919.637,E2 -14919.637} C_VEL
LIN {X 0,Y 339.162,Z 552.011,A -85,B 0,C 180,E1 -14920.952,E2 -14920.952} C_VEL
LIN {X 0,Y 337.557,Z 561.571,A -85,B 0,C 180,E1 -14922.429,E2 -14922.429} C_VEL
LIN {X 0,Y 335.716,Z 570.783,A -85,B 0,C 180,E1 -14924.208,E2 -14924.208} C_VEL
LIN {X 0,Y 333.971,Z 578.228,A -85,B 0,C 180,E1 -14925.995,E2 -14925.995} C_VEL
LIN {X 0,Y 332.49,Z 584.079,A -85,B 0,C 180,E1 -14927.797,E2 -14927.797} C_VEL
LIN {X 0,Y 331.161,Z 588.604,A -85,B 0,C 180,E1 -14929.608,E2 -14929.608} C_VEL
LIN {X 0,Y 329.994,Z 592.008,A -85,B 0,C 180,E1 -14931.426,E2 -14931.426} C_VEL
LIN {X 0,Y 329.286,Z 593.688,A -85,B 0,C 180,E1 -14932.643,E2 -14932.643} C_VEL
LIN {X 0,Y 328.765,Z 594.912,A -85,B 0,C 180,E1 -14933.864,E2 -14933.864} C_VEL
LIN {X 0,Y 328.417,Z 595.643,A -85,B 0,C 180,E1 -14935.09,E2 -14935.09} C_VEL
LIN {X 0,Y 327.995,Z 595.969,A -85,B 0,C 180,E1 -14936.314,E2 -14936.314} C_VEL
LIN {X 0,Y 327.626,Z 595.885,A -85,B 0,C 180,E1 -14937.541,E2 -14937.541} C_VEL
LIN {X 0,Y 327.31,Z 595.362,A -85,B 0,C 180,E1 -14938.77,E2 -14938.77} C_VEL
LIN {X 0,Y 326.951,Z 594.397,A -85,B 0,C 180,E1 -14940,E2 -14940} C_VEL
LIN {X 0,Y 326.958,Z 592.979,A -85,B 0,C 180,E1 -14941.232,E2 -14941.232} C_VEL
LIN {X 0,Y 326.85,Z 590.028,A -85,B 0,C 180,E1 -14943.082,E2 -14943.082} C_VEL
LIN {X 0,Y 326.802,Z 586.01,A -85,B 0,C 180,E1 -14944.935,E2 -14944.935} C_VEL
LIN {X 0,Y 327.187,Z 579.783,A -85,B 0,C 180,E1 -14947.095,E2 -14947.095} C_VEL
LIN {X 0,Y 327.647,Z 572.608,A -85,B 0,C 180,E1 -14949.043,E2 -14949.043} C_VEL
LIN {X 0,Y 327.99,Z 564.591,A -85,B 0,C 180,E1 -14950.806,E2 -14950.806} C_VEL
LIN {X 0,Y 328.639,Z 554.098,A -85,B 0,C 180,E1 -14952.662,E2 -14952.662} C_VEL
LIN {X 0,Y 329.215,Z 543.212,A -85,B 0,C 180,E1 -14954.211,E2 -14954.211} C_VEL
LIN {X 0,Y 329.914,Z 531.033,A -85,B 0,C 180,E1 -14955.602,E2 -14955.602} C_VEL
LIN {X 0,Y 330.437,Z 518.064,A -85,B 0,C 180,E1 -14956.758,E2 -14956.758} C_VEL
LIN {X 0,Y 330.821,Z 505.518,A -85,B 0,C 180,E1 -14957.622,E2 -14957.622} C_VEL
LIN {X 0,Y 331.136,Z 492.196,A -85,B 0,C 180,E1 -14958.283,E2 -14958.283} C_VEL
LIN {X 0,Y 331.359,Z 470.116,A -85,B 0,C 180,E1 -14958.992,E2 -14958.992} C_VEL
LIN {X 0,Y 332.439,Z 426.684,A -85,B 0,C 180,E1 -14960.285,E2 -14960.285} C_VEL
LIN {X 0,Y 326.896,Z 408.699,A -85,B 0,C 180,E1 -14961.087,E2 -14961.087} C_VEL
LIN {X 0,Y 326.721,Z 407.866,A -85,B 0,C 180,E1 -14961.322,E2 -14961.322} C_VEL
LIN {X 0,Y 326.64,Z 407.797,A -85,B 0,C 180,E1 -14965.488,E2 -14965.488} C_VEL
LIN {X 0,Y 326.623,Z 407.783,A -85,B 0,C 180,E1 -14968.254,E2 -14968.254} C_VEL
LIN {X 0,Y 326.576,Z 407.807,A -85,B 0,C 180,E1 -14971.097,E2 -14971.097} C_VEL
LIN {X 0,Y 326.609,Z 407.785,A -85,B 0,C 180,E1 -14974.019,E2 -14974.019} C_VEL
LIN {X 0,Y 326.629,Z 407.793,A -85,B 0,C 180,E1 -14977.239,E2 -14977.239} C_VEL
LIN {X 0,Y 326.579,Z 407.801,A -85,B 0,C 180,E1 -14981.131,E2 -14981.131} C_VEL
LIN {X 0,Y 326.529,Z 407.806,A -85,B 0,C 180,E1 -14984.743,E2 -14984.743} C_VEL
LIN {X 0,Y 326.576,Z 407.8,A -85,B 0,C 180,E1 -14988.154,E2 -14988.154} C_VEL
LIN {X 0,Y 326.654,Z 407.986,A -85,B 0,C 180,E1 -14991.281,E2 -14991.281} C_VEL
LIN {X 0,Y 331.022,Z 421.92,A -85,B 0,C 180,E1 -14994.31,E2 -14994.31} C_VEL
LIN {X 0,Y 334.549,Z 435.806,A -85,B 0,C 180,E1 -14997.172,E2 -14997.172} C_VEL
LIN {X 0,Y 336.488,Z 444.693,A -85,B 0,C 180,E1 -14998.909,E2 -14998.909} C_VEL
LIN {X 0,Y 335.927,Z 453.521,A -85,B 0,C 180,E1 -15000.379,E2 -15000.379} C_VEL
LIN {X 0,Y 333.973,Z 477.098,A -85,B 0,C 180,E1 -15004.11,E2 -15004.11} C_VEL
LIN {X 0,Y 333.204,Z 488.045,A -85,B 0,C 180,E1 -15005.759,E2 -15005.759} C_VEL
LIN {X 0,Y 337.404,Z 517.308,A -85,B 0,C 180,E1 -15006.758,E2 -15006.758} C_VEL
LIN {X 0,Y 336.151,Z 583.59,A -85,B 0,C 180,E1 -15008.176,E2 -15008.176} C_VEL
LIN {X 0,Y 335.64,Z 602.458,A -85,B 0,C 180,E1 -15008.625,E2 -15008.625} C_VEL
LIN {X 0,Y 334.804,Z 616.214,A -85,B 0,C 180,E1 -15009.214,E2 -15009.214} C_VEL
LIN {X 0,Y 333.913,Z 628.602,A -85,B 0,C 180,E1 -15010,E2 -15010} C_VEL
LIN {X 0,Y 332.571,Z 640.785,A -85,B 0,C 180,E1 -15011.04,E2 -15011.04} C_VEL
LIN {X 0,Y 331.283,Z 651.696,A -85,B 0,C 180,E1 -15012.244,E2 -15012.244} C_VEL
LIN {X 0,Y 330.067,Z 662.044,A -85,B 0,C 180,E1 -15013.69,E2 -15013.69} C_VEL
LIN {X 0,Y 328.926,Z 670.499,A -85,B 0,C 180,E1 -15015.144,E2 -15015.144} C_VEL
LIN {X 0,Y 327.608,Z 679.198,A -85,B 0,C 180,E1 -15016.982,E2 -15016.982} C_VEL
LIN {X 0,Y 326.647,Z 686.181,A -85,B 0,C 180,E1 -15018.835,E2 -15018.835} C_VEL
LIN {X 0,Y 325.902,Z 691.73,A -85,B 0,C 180,E1 -15020.692,E2 -15020.692} C_VEL
LIN {X 0,Y 325.448,Z 696.085,A -85,B 0,C 180,E1 -15022.555,E2 -15022.555} C_VEL
LIN {X 0,Y 325.194,Z 698.378,A -85,B 0,C 180,E1 -15023.797,E2 -15023.797} C_VEL
LIN {X 0,Y 325.03,Z 700.247,A -85,B 0,C 180,E1 -15025.038,E2 -15025.038} C_VEL
LIN {X 0,Y 324.94,Z 701.674,A -85,B 0,C 180,E1 -15026.28,E2 -15026.28} C_VEL
LIN {X 0,Y 324.788,Z 703.292,A -85,B 0,C 180,E1 -15028.76,E2 -15028.76} C_VEL
LIN {X 0,Y 324.794,Z 703.527,A -85,B 0,C 180,E1 -15030,E2 -15030} C_VEL
LIN {X 0,Y 324.788,Z 703.332,A -85,B 0,C 180,E1 -15031.24,E2 -15031.24} C_VEL
LIN {X 0,Y 324.938,Z 701.767,A -85,B 0,C 180,E1 -15033.721,E2 -15033.721} C_VEL
LIN {X 0,Y 325.016,Z 700.392,A -85,B 0,C 180,E1 -15034.962,E2 -15034.962} C_VEL
LIN {X 0,Y 325.26,Z 697.503,A -85,B 0,C 180,E1 -15036.825,E2 -15036.825} C_VEL
LIN {X 0,Y 325.677,Z 693.578,A -85,B 0,C 180,E1 -15038.688,E2 -15038.688} C_VEL
LIN {X 0,Y 326.306,Z 688.493,A -85,B 0,C 180,E1 -15040.549,E2 -15040.549} C_VEL
LIN {X 0,Y 327.174,Z 682.083,A -85,B 0,C 180,E1 -15042.405,E2 -15042.405} C_VEL
LIN {X 0,Y 328.402,Z 674.121,A -85,B 0,C 180,E1 -15044.248,E2 -15044.248} C_VEL
LIN {X 0,Y 329.587,Z 665.984,A -85,B 0,C 180,E1 -15045.776,E2 -15045.776} C_VEL
LIN {X 0,Y 330.782,Z 655.975,A -85,B 0,C 180,E1 -15047.305,E2 -15047.305} C_VEL
LIN {X 0,Y 332.167,Z 644.723,A -85,B 0,C 180,E1 -15048.664,E2 -15048.664} C_VEL
LIN {X 0,Y 333.458,Z 633.679,A -85,B 0,C 180,E1 -15049.708,E2 -15049.708} C_VEL
LIN {X 0,Y 334.472,Z 621.202,A -85,B 0,C 180,E1 -15050.607,E2 -15050.607} C_VEL
LIN {X 0,Y 335.383,Z 608.152,A -85,B 0,C 180,E1 -15051.272,E2 -15051.272} C_VEL
LIN {X 0,Y 335.983,Z 595.315,A -85,B 0,C 180,E1 -15051.675,E2 -15051.675} C_VEL
LIN {X 0,Y 336.512,Z 567.246,A -85,B 0,C 180,E1 -15052.278,E2 -15052.278} C_VEL
LIN {X 0,Y 335.991,Z 561.438,A -85,B 0,C 180,E1 -15052.446,E2 -15052.446} C_VEL
LIN {X 0,Y 331.035,Z 542.765,A -85,B 0,C 180,E1 -15053.233,E2 -15053.233} C_VEL
LIN {X 0,Y 330.571,Z 536.956,A -85,B 0,C 180,E1 -15053.402,E2 -15053.402} C_VEL
LIN {X 0,Y 330.904,Z 518.175,A -85,B 0,C 180,E1 -15053.815,E2 -15053.815} C_VEL
LIN {X 0,Y 326.83,Z 489.334,A -85,B 0,C 180,E1 -15054.814,E2 -15054.814} C_VEL
LIN {X 0,Y 326.634,Z 487.659,A -85,B 0,C 180,E1 -15054.908,E2 -15054.908} C_VEL
LIN {X 0,Y 328.324,Z 466.155,A -85,B 0,C 180,E1 -15058.286,E2 -15058.286} C_VEL
LIN {X 0,Y 329.927,Z 448.283,A -85,B 0,C 180,E1 -15061.204,E2 -15061.204} C_VEL
LIN {X 0,Y 329.47,Z 444.622,A -85,B 0,C 180,E1 -15061.902,E2 -15061.902} C_VEL
LIN {X 0,Y 326.277,Z 430.946,A -85,B 0,C 180,E1 -15064.684,E2 -15064.684} C_VEL
LIN {X 0,Y 322.332,Z 417.14,A -85,B 0,C 180,E1 -15067.626,E2 -15067.626} C_VEL
LIN {X 0,Y 319.547,Z 408.851,A -85,B 0,C 180,E1 -15069.56,E2 -15069.56} C_VEL
LIN {X 0,Y 319.522,Z 408.667,A -85,B 0,C 180,E1 -15073.46,E2 -15073.46} C_VEL
LIN {X 0,Y 319.554,Z 408.681,A -85,B 0,C 180,E1 -15077.016,E2 -15077.016} C_VEL
LIN {X 0,Y 319.547,Z 408.682,A -85,B 0,C 180,E1 -15080.371,E2 -15080.371} C_VEL
LIN {X 0,Y 319.581,Z 408.677,A -85,B 0,C 180,E1 -15084.458,E2 -15084.458} C_VEL
LIN {X 0,Y 319.527,Z 408.683,A -85,B 0,C 180,E1 -15088.137,E2 -15088.137} C_VEL
LIN {X 0,Y 319.547,Z 408.668,A -85,B 0,C 180,E1 -15091.613,E2 -15091.613} C_VEL
LIN {X 0,Y 319.574,Z 408.668,A -85,B 0,C 180,E1 -15095.301,E2 -15095.301} C_VEL
LIN {X 0,Y 319.567,Z 408.673,A -85,B 0,C 180,E1 -15098.045,E2 -15098.045} C_VEL
LIN {X 0,Y 319.59,Z 408.655,A -85,B 0,C 180,E1 -15102.069,E2 -15102.069} C_VEL
LIN {X 0,Y 319.712,Z 408.658,A -85,B 0,C 180,E1 -15106.007,E2 -15106.007} C_VEL
LIN {X 0,Y 319.737,Z 408.64,A -85,B 0,C 180,E1 -15109.872,E2 -15109.872} C_VEL
LIN {X 0,Y 319.901,Z 408.625,A -85,B 0,C 180,E1 -15113.693,E2 -15113.693} C_VEL
LIN {X 0,Y 319.957,Z 408.621,A -85,B 0,C 180,E1 -15117.482,E2 -15117.482} C_VEL
LIN {X 0,Y 320,Z 408.606,A -85,B 0,C 180,E1 -15121.258,E2 -15121.258} C_VEL
LIN {X 0,Y 319.693,Z 408.643,A -85,B 0,C 180,E1 -15123.781,E2 -15123.781} C_VEL
LIN {X 0,Y 319.903,Z 408.636,A -85,B 0,C 180,E1 -15126.306,E2 -15126.306} C_VEL
LIN {X 0,Y 319.737,Z 408.633,A -85,B 0,C 180,E1 -15130.128,E2 -15130.128} C_VEL
LIN {X 0,Y 319.703,Z 408.658,A -85,B 0,C 180,E1 -15133.993,E2 -15133.993} C_VEL
LIN {X 0,Y 319.574,Z 408.662,A -85,B 0,C 180,E1 -15137.932,E2 -15137.932} C_VEL
LIN {X 0,Y 319.564,Z 408.663,A -85,B 0,C 180,E1 -15141.955,E2 -15141.955} C_VEL
LIN {X 0,Y 319.552,Z 408.681,A -85,B 0,C 180,E1 -15146.095,E2 -15146.095} C_VEL
LIN {X 0,Y 319.527,Z 408.663,A -85,B 0,C 180,E1 -15148.94,E2 -15148.94} C_VEL
LIN {X 0,Y 319.527,Z 408.686,A -85,B 0,C 180,E1 -15151.862,E2 -15151.862} C_VEL
LIN {X 0,Y 319.58,Z 408.667,A -85,B 0,C 180,E1 -15155.542,E2 -15155.542} C_VEL
LIN {X 0,Y 319.525,Z 408.677,A -85,B 0,C 180,E1 -15158.015,E2 -15158.015} C_VEL
LIN {X 0,Y 319.504,Z 408.631,A -85,B 0,C 180,E1 -15161.592,E2 -15161.592} C_VEL
LIN {X 0,Y 319.487,Z 408.687,A -85,B 0,C 180,E1 -15164.743,E2 -15164.743} C_VEL
LIN {X 0,Y 319.551,Z 408.66,A -85,B 0,C 180,E1 -15167.016,E2 -15167.016} C_VEL
LIN {X 0,Y 319.516,Z 408.655,A -85,B 0,C 180,E1 -15170.366,E2 -15170.366} C_VEL
LIN {X 0,Y 319.654,Z 408.871,A -85,B 0,C 180,E1 -15173.926,E2 -15173.926} C_VEL
LIN {X 0,Y 323.077,Z 424.977,A -85,B 0,C 180,E1 -15177.561,E2 -15177.561} C_VEL
LIN {X 0,Y 325.459,Z 435.965,A -85,B 0,C 180,E1 -15179.946,E2 -15179.946} C_VEL
LIN {X 0,Y 324.148,Z 447.872,A -85,B 0,C 180,E1 -15182.285,E2 -15182.285} C_VEL
LIN {X 0,Y 325.965,Z 478.487,A -85,B 0,C 180,E1 -15184.55,E2 -15184.55} C_VEL
LIN {X 0,Y 326.382,Z 488.487,A -85,B 0,C 180,E1 -15185.305,E2 -15185.305} C_VEL
LIN {X 0,Y 329.629,Z 517.982,A -85,B 0,C 180,E1 -15186.255,E2 -15186.255} C_VEL
LIN {X 0,Y 330.347,Z 526.427,A -85,B 0,C 180,E1 -15186.505,E2 -15186.505} C_VEL
LIN {X 0,Y 328.702,Z 603.966,A -85,B 0,C 180,E1 -15188.192,E2 -15188.192} C_VEL
LIN {X 0,Y 327.968,Z 617.352,A -85,B 0,C 180,E1 -15188.677,E2 -15188.677} C_VEL
LIN {X 0,Y 327.038,Z 629.864,A -85,B 0,C 180,E1 -15189.396,E2 -15189.396} C_VEL
LIN {X 0,Y 325.938,Z 641.523,A -85,B 0,C 180,E1 -15190.311,E2 -15190.311} C_VEL
LIN {X 0,Y 324.682,Z 652.13,A -85,B 0,C 180,E1 -15191.381,E2 -15191.381} C_VEL
LIN {X 0,Y 323.304,Z 662.938,A -85,B 0,C 180,E1 -15192.772,E2 -15192.772} C_VEL
LIN {X 0,Y 321.895,Z 673.495,A -85,B 0,C 180,E1 -15194.487,E2 -15194.487} C_VEL
LIN {X 0,Y 320.603,Z 682.602,A -85,B 0,C 180,E1 -15196.37,E2 -15196.37} C_VEL
LIN {X 0,Y 319.551,Z 689.913,A -85,B 0,C 180,E1 -15198.262,E2 -15198.262} C_VEL
LIN {X 0,Y 318.712,Z 696.602,A -85,B 0,C 180,E1 -15200.48,E2 -15200.48} C_VEL
LIN {X 0,Y 318.224,Z 700.989,A -85,B 0,C 180,E1 -15202.385,E2 -15202.385} C_VEL
LIN {X 0,Y 318.004,Z 703.865,A -85,B 0,C 180,E1 -15203.997,E2 -15203.997} C_VEL
LIN {X 0,Y 317.875,Z 706.597,A -85,B 0,C 180,E1 -15206.197,E2 -15206.197} C_VEL
LIN {X 0,Y 317.813,Z 707.597,A -85,B 0,C 180,E1 -15207.465,E2 -15207.465} C_VEL
LIN {X 0,Y 317.766,Z 708.208,A -85,B 0,C 180,E1 -15208.733,E2 -15208.733} C_VEL
LIN {X 0,Y 317.794,Z 708.425,A -85,B 0,C 180,E1 -15210,E2 -15210} C_VEL
LIN {X 0,Y 317.8,Z 708.202,A -85,B 0,C 180,E1 -15211.267,E2 -15211.267} C_VEL
LIN {X 0,Y 317.9,Z 706.584,A -85,B 0,C 180,E1 -15213.803,E2 -15213.803} C_VEL
LIN {X 0,Y 318.01,Z 703.824,A -85,B 0,C 180,E1 -15216.012,E2 -15216.012} C_VEL
LIN {X 0,Y 318.359,Z 699.609,A -85,B 0,C 180,E1 -15218.25,E2 -15218.25} C_VEL
LIN {X 0,Y 318.924,Z 694.815,A -85,B 0,C 180,E1 -15220.154,E2 -15220.154} C_VEL
LIN {X 0,Y 319.692,Z 688.747,A -85,B 0,C 180,E1 -15222.055,E2 -15222.055} C_VEL
LIN {X 0,Y 320.792,Z 681.177,A -85,B 0,C 180,E1 -15223.945,E2 -15223.945} C_VEL
LIN {X 0,Y 321.897,Z 673.389,A -85,B 0,C 180,E1 -15225.513,E2 -15225.513} C_VEL
LIN {X 0,Y 323.277,Z 662.809,A -85,B 0,C 180,E1 -15227.229,E2 -15227.229} C_VEL
LIN {X 0,Y 324.662,Z 651.968,A -85,B 0,C 180,E1 -15228.62,E2 -15228.62} C_VEL
LIN {X 0,Y 325.929,Z 641.319,A -85,B 0,C 180,E1 -15229.689,E2 -15229.689} C_VEL
LIN {X 0,Y 327.028,Z 629.6,A -85,B 0,C 180,E1 -15230.604,E2 -15230.604} C_VEL
LIN {X 0,Y 327.976,Z 616.96,A -85,B 0,C 180,E1 -15231.322,E2 -15231.322} C_VEL
LIN {X 0,Y 328.295,Z 613.514,A -85,B 0,C 180,E1 -15231.506,E2 -15231.506} C_VEL
LIN {X 0,Y 330.777,Z 600.459,A -85,B 0,C 180,E1 -15232.65,E2 -15232.65} C_VEL
LIN {X 0,Y 333.112,Z 585.84,A -85,B 0,C 180,E1 -15233.632,E2 -15233.632} C_VEL
LIN {X 0,Y 334.791,Z 571.663,A -85,B 0,C 180,E1 -15234.329,E2 -15234.329} C_VEL
LIN {X 0,Y 338.049,Z 526.631,A -85,B 0,C 180,E1 -15235.946,E2 -15235.946} C_VEL
LIN {X 0,Y 337.805,Z 508.853,A -85,B 0,C 180,E1 -15236.834,E2 -15236.834} C_VEL
LIN {X 0,Y 336.661,Z 492.76,A -85,B 0,C 180,E1 -15237.836,E2 -15237.836} C_VEL
LIN {X 0,Y 334.813,Z 477.235,A -85,B 0,C 180,E1 -15239.006,E2 -15239.006} C_VEL
LIN {X 0,Y 332.527,Z 462.607,A -85,B 0,C 180,E1 -15240.321,E2 -15240.321} C_VEL
LIN {X 0,Y 330.892,Z 453.572,A -85,B 0,C 180,E1 -15241.253,E2 -15241.253} C_VEL
LIN {X 0,Y 330.487,Z 449.961,A -85,B 0,C 180,E1 -15241.655,E2 -15241.655} C_VEL
LIN {X 0,Y 330.651,Z 448.178,A -85,B 0,C 180,E1 -15242.098,E2 -15242.098} C_VEL
LIN {X 0,Y 329.467,Z 441.101,A -85,B 0,C 180,E1 -15244.421,E2 -15244.421} C_VEL
LIN {X 0,Y 327.985,Z 434.707,A -85,B 0,C 180,E1 -15246.868,E2 -15246.868} C_VEL
LIN {X 0,Y 326.12,Z 427.953,A -85,B 0,C 180,E1 -15249.995,E2 -15249.995} C_VEL
LIN {X 0,Y 324.65,Z 423.54,A -85,B 0,C 180,E1 -15252.606,E2 -15252.606} C_VEL
LIN {X 0,Y 323.173,Z 419.307,A -85,B 0,C 180,E1 -15255.901,E2 -15255.901} C_VEL
LIN {X 0,Y 322.199,Z 416.531,A -85,B 0,C 180,E1 -15259.127,E2 -15259.127} C_VEL
LIN {X 0,Y 321.703,Z 415.025,A -85,B 0,C 180,E1 -15262.288,E2 -15262.288} C_VEL
LIN {X 0,Y 321.62,Z 414.691,A -85,B 0,C 180,E1 -15263.952,E2 -15263.952} C_VEL
LIN {X 0,Y 321.724,Z 414.965,A -85,B 0,C 180,E1 -15265.737,E2 -15265.737} C_VEL
LIN {X 0,Y 324.597,Z 417.754,A -85,B 0,C 180,E1 -15267.229,E2 -15267.229} C_VEL
LIN {X 0,Y 328.633,Z 421.867,A -85,B 0,C 180,E1 -15268.887,E2 -15268.887} C_VEL
LIN {X 0,Y 330.972,Z 424.838,A -85,B 0,C 180,E1 -15269.768,E2 -15269.768} C_VEL
LIN {X 0,Y 334.117,Z 429.82,A -85,B 0,C 180,E1 -15270.921,E2 -15270.921} C_VEL
LIN {X 0,Y 337.917,Z 435.861,A -85,B 0,C 180,E1 -15272.15,E2 -15272.15} C_VEL
LIN {X 0,Y 342.526,Z 444.677,A -85,B 0,C 180,E1 -15273.564,E2 -15273.564} C_VEL
LIN {X 0,Y 343.181,Z 446.173,A -85,B 0,C 180,E1 -15273.769,E2 -15273.769} C_VEL
LIN {X 0,Y 339.604,Z 487.446,A -85,B 0,C 180,E1 -15275.285,E2 -15275.285} C_VEL
LIN {X 0,Y 338.602,Z 506.691,A -85,B 0,C 180,E1 -15276.12,E2 -15276.12} C_VEL
LIN {X 0,Y 337.645,Z 520.261,A -85,B 0,C 180,E1 -15276.947,E2 -15276.947} C_VEL
LIN {X 0,Y 336.427,Z 532.212,A -85,B 0,C 180,E1 -15277.912,E2 -15277.912} C_VEL
LIN {X 0,Y 334.888,Z 543.761,A -85,B 0,C 180,E1 -15279.098,E2 -15279.098} C_VEL
LIN {X 0,Y 333.107,Z 554.119,A -85,B 0,C 180,E1 -15280.431,E2 -15280.431} C_VEL
LIN {X 0,Y 331.231,Z 564.378,A -85,B 0,C 180,E1 -15282.082,E2 -15282.082} C_VEL
LIN {X 0,Y 329.276,Z 573.283,A -85,B 0,C 180,E1 -15283.891,E2 -15283.891} C_VEL
LIN {X 0,Y 327.42,Z 580.399,A -85,B 0,C 180,E1 -15285.709,E2 -15285.709} C_VEL
LIN {X 0,Y 325.815,Z 586.03,A -85,B 0,C 180,E1 -15287.543,E2 -15287.543} C_VEL
LIN {X 0,Y 324.429,Z 590.398,A -85,B 0,C 180,E1 -15289.389,E2 -15289.389} C_VEL
LIN {X 0,Y 323.185,Z 593.629,A -85,B 0,C 180,E1 -15291.244,E2 -15291.244} C_VEL
LIN {X 0,Y 322.43,Z 595.21,A -85,B 0,C 180,E1 -15292.485,E2 -15292.485} C_VEL
LIN {X 0,Y 321.858,Z 596.305,A -85,B 0,C 180,E1 -15293.732,E2 -15293.732} C_VEL
LIN {X 0,Y 321.483,Z 596.94,A -85,B 0,C 180,E1 -15294.983,E2 -15294.983} C_VEL
LIN {X 0,Y 321.044,Z 597.188,A -85,B 0,C 180,E1 -15296.235,E2 -15296.235} C_VEL
LIN {X 0,Y 320.625,Z 597.014,A -85,B 0,C 180,E1 -15297.487,E2 -15297.487} C_VEL
LIN {X 0,Y 320.307,Z 596.365,A -85,B 0,C 180,E1 -15298.743,E2 -15298.743} C_VEL
LIN {X 0,Y 319.923,Z 595.321,A -85,B 0,C 180,E1 -15300,E2 -15300} C_VEL
LIN {X 0,Y 319.93,Z 593.812,A -85,B 0,C 180,E1 -15301.259,E2 -15301.259} C_VEL
LIN {X 0,Y 319.81,Z 590.711,A -85,B 0,C 180,E1 -15303.149,E2 -15303.149} C_VEL
LIN {X 0,Y 319.76,Z 586.521,A -85,B 0,C 180,E1 -15305.044,E2 -15305.044} C_VEL
LIN {X 0,Y 320.148,Z 580.065,A -85,B 0,C 180,E1 -15307.252,E2 -15307.252} C_VEL
LIN {X 0,Y 320.588,Z 573.122,A -85,B 0,C 180,E1 -15309.133,E2 -15309.133} C_VEL
LIN {X 0,Y 320.976,Z 564.352,A -85,B 0,C 180,E1 -15311.046,E2 -15311.046} C_VEL
LIN {X 0,Y 321.547,Z 555.494,A -85,B 0,C 180,E1 -15312.625,E2 -15312.625} C_VEL
LIN {X 0,Y 322.133,Z 544.684,A -85,B 0,C 180,E1 -15314.208,E2 -15314.208} C_VEL
LIN {X 0,Y 322.824,Z 532.585,A -85,B 0,C 180,E1 -15315.629,E2 -15315.629} C_VEL
LIN {X 0,Y 323.351,Z 521.005,A -85,B 0,C 180,E1 -15316.717,E2 -15316.717} C_VEL
LIN {X 0,Y 323.748,Z 507.582,A -85,B 0,C 180,E1 -15317.693,E2 -15317.693} C_VEL
LIN {X 0,Y 324.113,Z 494.073,A -85,B 0,C 180,E1 -15318.407,E2 -15318.407} C_VEL
LIN {X 0,Y 324.335,Z 473.098,A -85,B 0,C 180,E1 -15319.121,E2 -15319.121} C_VEL
LIN {X 0,Y 325.486,Z 428.065,A -85,B 0,C 180,E1 -15320.504,E2 -15320.504} C_VEL
LIN {X 0,Y 319.794,Z 409.448,A -85,B 0,C 180,E1 -15321.366,E2 -15321.366} C_VEL
LIN {X 0,Y 319.648,Z 408.715,A -85,B 0,C 180,E1 -15321.645,E2 -15321.645} C_VEL
LIN {X 0,Y 319.575,Z 408.677,A -85,B 0,C 180,E1 -15326.093,E2 -15326.093} C_VEL
LIN {X 0,Y 319.554,Z 408.661,A -85,B 0,C 180,E1 -15328.937,E2 -15328.937} C_VEL
LIN {X 0,Y 319.526,Z 408.683,A -85,B 0,C 180,E1 -15331.863,E2 -15331.863} C_VEL
LIN {X 0,Y 319.582,Z 408.676,A -85,B 0,C 180,E1 -15335.543,E2 -15335.543} C_VEL
LIN {X 0,Y 319.56,Z 408.679,A -85,B 0,C 180,E1 -15339.669,E2 -15339.669} C_VEL
LIN {X 0,Y 319.523,Z 408.686,A -85,B 0,C 180,E1 -15343.461,E2 -15343.461} C_VEL
LIN {X 0,Y 319.555,Z 408.68,A -85,B 0,C 180,E1 -15347.017,E2 -15347.017} C_VEL
LIN {X 0,Y 319.591,Z 408.844,A -85,B 0,C 180,E1 -15350.569,E2 -15350.569} C_VEL
LIN {X 0,Y 323.681,Z 421.657,A -85,B 0,C 180,E1 -15353.454,E2 -15353.454} C_VEL
LIN {X 0,Y 326.916,Z 433.7,A -85,B 0,C 180,E1 -15356.017,E2 -15356.017} C_VEL
LIN {X 0,Y 329.725,Z 445.997,A -85,B 0,C 180,E1 -15358.495,E2 -15358.495} C_VEL
LIN {X 0,Y 329.832,Z 449.079,A -85,B 0,C 180,E1 -15359.041,E2 -15359.041} C_VEL
LIN {X 0,Y 327.885,Z 470.675,A -85,B 0,C 180,E1 -15362.559,E2 -15362.559} C_VEL
LIN {X 0,Y 326.6,Z 488.053,A -85,B 0,C 180,E1 -15365.238,E2 -15365.238} C_VEL
LIN {X 0,Y 330.887,Z 518.31,A -85,B 0,C 180,E1 -15366.297,E2 -15366.297} C_VEL
LIN {X 0,Y 329.273,Z 597.318,A -85,B 0,C 180,E1 -15368.026,E2 -15368.026} C_VEL
LIN {X 0,Y 328.549,Z 610.956,A -85,B 0,C 180,E1 -15368.511,E2 -15368.511} C_VEL
LIN {X 0,Y 327.707,Z 623.254,A -85,B 0,C 180,E1 -15369.194,E2 -15369.194} C_VEL
LIN {X 0,Y 326.62,Z 634.287,A -85,B 0,C 180,E1 -15370.026,E2 -15370.026} C_VEL
LIN {X 0,Y 325.393,Z 645.219,A -85,B 0,C 180,E1 -15371.096,E2 -15371.096} C_VEL
LIN {X 0,Y 324.116,Z 655.249,A -85,B 0,C 180,E1 -15372.328,E2 -15372.328} C_VEL
LIN {X 0,Y 322.826,Z 665.427,A -85,B 0,C 180,E1 -15373.885,E2 -15373.885} C_VEL
LIN {X 0,Y 321.348,Z 675.136,A -85,B 0,C 180,E1 -15375.757,E2 -15375.757} C_VEL
LIN {X 0,Y 320.146,Z 682.94,A -85,B 0,C 180,E1 -15377.641,E2 -15377.641} C_VEL
LIN {X 0,Y 319.371,Z 688.214,A -85,B 0,C 180,E1 -15379.22,E2 -15379.22} C_VEL
LIN {X 0,Y 318.678,Z 693.367,A -85,B 0,C 180,E1 -15381.12,E2 -15381.12} C_VEL
LIN {X 0,Y 318.255,Z 697.358,A -85,B 0,C 180,E1 -15383.024,E2 -15383.024} C_VEL
LIN {X 0,Y 317.946,Z 700.302,A -85,B 0,C 180,E1 -15384.928,E2 -15384.928} C_VEL
LIN {X 0,Y 317.853,Z 701.729,A -85,B 0,C 180,E1 -15386.197,E2 -15386.197} C_VEL
LIN {X 0,Y 317.766,Z 702.729,A -85,B 0,C 180,E1 -15387.465,E2 -15387.465} C_VEL
LIN {X 0,Y 317.705,Z 703.581,A -85,B 0,C 180,E1 -15390,E2 -15390} C_VEL
LIN {X 0,Y 317.703,Z 703.386,A -85,B 0,C 180,E1 -15391.268,E2 -15391.268} C_VEL
LIN {X 0,Y 317.765,Z 702.795,A -85,B 0,C 180,E1 -15392.535,E2 -15392.535} C_VEL
LIN {X 0,Y 317.85,Z 701.821,A -85,B 0,C 180,E1 -15393.804,E2 -15393.804} C_VEL
LIN {X 0,Y 318.037,Z 699.077,A -85,B 0,C 180,E1 -15396.056,E2 -15396.056} C_VEL
LIN {X 0,Y 318.46,Z 695.037,A -85,B 0,C 180,E1 -15398.248,E2 -15398.248} C_VEL
LIN {X 0,Y 319.082,Z 690.354,A -85,B 0,C 180,E1 -15400.149,E2 -15400.149} C_VEL
LIN {X 0,Y 320.072,Z 683.323,A -85,B 0,C 180,E1 -15402.362,E2 -15402.362} C_VEL
LIN {X 0,Y 321.303,Z 675.619,A -85,B 0,C 180,E1 -15404.246,E2 -15404.246} C_VEL
LIN {X 0,Y 322.529,Z 667.766,A -85,B 0,C 180,E1 -15405.806,E2 -15405.806} C_VEL
LIN {X 0,Y 323.706,Z 658.297,A -85,B 0,C 180,E1 -15407.353,E2 -15407.353} C_VEL
LIN {X 0,Y 324.955,Z 648.828,A -85,B 0,C 180,E1 -15408.603,E2 -15408.603} C_VEL
LIN {X 0,Y 326.174,Z 638.788,A -85,B 0,C 180,E1 -15409.674,E2 -15409.674} C_VEL
LIN {X 0,Y 327.362,Z 626.867,A -85,B 0,C 180,E1 -15410.664,E2 -15410.664} C_VEL
LIN {X 0,Y 328.422,Z 613.869,A -85,B 0,C 180,E1 -15411.457,E2 -15411.457} C_VEL
LIN {X 0,Y 329.18,Z 600.795,A -85,B 0,C 180,E1 -15411.981,E2 -15411.981} C_VEL
LIN {X 0,Y 330.576,Z 537.972,A -85,B 0,C 180,E1 -15413.378,E2 -15413.378} C_VEL
LIN {X 0,Y 330.571,Z 536.956,A -85,B 0,C 180,E1 -15413.402,E2 -15413.402} C_VEL
LIN {X 0,Y 330.05,Z 531.146,A -85,B 0,C 180,E1 -15413.577,E2 -15413.577} C_VEL
LIN {X 0,Y 327.261,Z 521.918,A -85,B 0,C 180,E1 -15414.007,E2 -15414.007} C_VEL
LIN {X 0,Y 323.558,Z 510.863,A -85,B 0,C 180,E1 -15414.563,E2 -15414.563} C_VEL
LIN {X 0,Y 322.877,Z 507.001,A -85,B 0,C 180,E1 -15414.711,E2 -15414.711} C_VEL
LIN {X 0,Y 320.068,Z 487.773,A -85,B 0,C 180,E1 -15415.44,E2 -15415.44} C_VEL
LIN {X 0,Y 321.837,Z 465.905,A -85,B 0,C 180,E1 -15418.92,E2 -15418.92} C_VEL
LIN {X 0,Y 323.317,Z 449.738,A -85,B 0,C 180,E1 -15421.597,E2 -15421.597} C_VEL
LIN {X 0,Y 321.407,Z 440.18,A -85,B 0,C 180,E1 -15423.532,E2 -15423.532} C_VEL
LIN {X 0,Y 318.11,Z 427.315,A -85,B 0,C 180,E1 -15426.255,E2 -15426.255} C_VEL
LIN {X 0,Y 314.821,Z 416.701,A -85,B 0,C 180,E1 -15428.617,E2 -15428.617} C_VEL
LIN {X 0,Y 312.475,Z 409.715,A -85,B 0,C 180,E1 -15430.314,E2 -15430.314} C_VEL
LIN {X 0,Y 312.452,Z 409.538,A -85,B 0,C 180,E1 -15434.21,E2 -15434.21} C_VEL
LIN {X 0,Y 312.458,Z 409.567,A -85,B 0,C 180,E1 -15437.925,E2 -15437.925} C_VEL
LIN {X 0,Y 312.486,Z 409.554,A -85,B 0,C 180,E1 -15441.923,E2 -15441.923} C_VEL
LIN {X 0,Y 312.533,Z 409.556,A -85,B 0,C 180,E1 -15444.22,E2 -15444.22} C_VEL
LIN {X 0,Y 312.504,Z 409.547,A -85,B 0,C 180,E1 -15447.334,E2 -15447.334} C_VEL
LIN {X 0,Y 312.488,Z 409.546,A -85,B 0,C 180,E1 -15451.299,E2 -15451.299} C_VEL
LIN {X 0,Y 312.549,Z 409.551,A -85,B 0,C 180,E1 -15454.708,E2 -15454.708} C_VEL
LIN {X 0,Y 312.522,Z 409.556,A -85,B 0,C 180,E1 -15458.911,E2 -15458.911} C_VEL
LIN {X 0,Y 312.554,Z 409.533,A -85,B 0,C 180,E1 -15461.651,E2 -15461.651} C_VEL
LIN {X 0,Y 312.654,Z 409.54,A -85,B 0,C 180,E1 -15465.684,E2 -15465.684} C_VEL
LIN {X 0,Y 312.687,Z 409.515,A -85,B 0,C 180,E1 -15469.641,E2 -15469.641} C_VEL
LIN {X 0,Y 312.799,Z 409.52,A -85,B 0,C 180,E1 -15472.252,E2 -15472.252} C_VEL
LIN {X 0,Y 312.688,Z 409.511,A -85,B 0,C 180,E1 -15474.842,E2 -15474.842} C_VEL
LIN {X 0,Y 312.971,Z 409.498,A -85,B 0,C 180,E1 -15478.713,E2 -15478.713} C_VEL
LIN {X 0,Y 312.969,Z 409.481,A -85,B 0,C 180,E1 -15481.287,E2 -15481.287} C_VEL
LIN {X 0,Y 312.691,Z 409.531,A -85,B 0,C 180,E1 -15485.158,E2 -15485.158} C_VEL
LIN {X 0,Y 312.799,Z 409.511,A -85,B 0,C 180,E1 -15487.748,E2 -15487.748} C_VEL
LIN {X 0,Y 312.661,Z 409.529,A -85,B 0,C 180,E1 -15491.672,E2 -15491.672} C_VEL
LIN {X 0,Y 312.607,Z 409.537,A -85,B 0,C 180,E1 -15494.821,E2 -15494.821} C_VEL
LIN {X 0,Y 312.537,Z 409.551,A -85,B 0,C 180,E1 -15499.185,E2 -15499.185} C_VEL
LIN {X 0,Y 312.516,Z 409.534,A -85,B 0,C 180,E1 -15502.775,E2 -15502.775} C_VEL
LIN {X 0,Y 312.485,Z 409.559,A -85,B 0,C 180,E1 -15506.732,E2 -15506.732} C_VEL
LIN {X 0,Y 312.471,Z 409.544,A -85,B 0,C 180,E1 -15509.658,E2 -15509.658} C_VEL
LIN {X 0,Y 312.522,Z 409.543,A -85,B 0,C 180,E1 -15513.688,E2 -15513.688} C_VEL
LIN {X 0,Y 312.512,Z 409.559,A -85,B 0,C 180,E1 -15517.387,E2 -15517.387} C_VEL
LIN {X 0,Y 312.441,Z 409.512,A -85,B 0,C 180,E1 -15520.717,E2 -15520.717} C_VEL
LIN {X 0,Y 312.451,Z 409.552,A -85,B 0,C 180,E1 -15524.21,E2 -15524.21} C_VEL
LIN {X 0,Y 312.455,Z 409.527,A -85,B 0,C 180,E1 -15527.925,E2 -15527.925} C_VEL
LIN {X 0,Y 312.485,Z 409.562,A -85,B 0,C 180,E1 -15531.922,E2 -15531.922} C_VEL
LIN {X 0,Y 312.623,Z 409.791,A -85,B 0,C 180,E1 -15533.682,E2 -15533.682} C_VEL
LIN {X 0,Y 316.223,Z 426.887,A -85,B 0,C 180,E1 -15537.623,E2 -15537.623} C_VEL
LIN {X 0,Y 318.455,Z 437.109,A -85,B 0,C 180,E1 -15539.878,E2 -15539.878} C_VEL
LIN {X 0,Y 317.631,Z 444.48,A -85,B 0,C 180,E1 -15541.368,E2 -15541.368} C_VEL
LIN {X 0,Y 317.875,Z 450.417,A -85,B 0,C 180,E1 -15541.867,E2 -15541.867} C_VEL
LIN {X 0,Y 319.319,Z 475.109,A -85,B 0,C 180,E1 -15543.721,E2 -15543.721} C_VEL
LIN {X 0,Y 319.857,Z 488.586,A -85,B 0,C 180,E1 -15544.768,E2 -15544.768} C_VEL
LIN {X 0,Y 323.138,Z 518.657,A -85,B 0,C 180,E1 -15545.762,E2 -15545.762} C_VEL
LIN {X 0,Y 323.818,Z 527.83,A -85,B 0,C 180,E1 -15546.034,E2 -15546.034} C_VEL
LIN {X 0,Y 322.118,Z 604.014,A -85,B 0,C 180,E1 -15547.722,E2 -15547.722} C_VEL
LIN {X 0,Y 321.37,Z 617.348,A -85,B 0,C 180,E1 -15548.217,E2 -15548.217} C_VEL
LIN {X 0,Y 320.404,Z 629.843,A -85,B 0,C 180,E1 -15548.95,E2 -15548.95} C_VEL
LIN {X 0,Y 319.269,Z 641.492,A -85,B 0,C 180,E1 -15549.882,E2 -15549.882} C_VEL
LIN {X 0,Y 317.962,Z 652.093,A -85,B 0,C 180,E1 -15550.972,E2 -15550.972} C_VEL
LIN {X 0,Y 316.512,Z 662.895,A -85,B 0,C 180,E1 -15552.39,E2 -15552.39} C_VEL
LIN {X 0,Y 315.231,Z 671.956,A -85,B 0,C 180,E1 -15553.87,E2 -15553.87} C_VEL
LIN {X 0,Y 313.893,Z 681.202,A -85,B 0,C 180,E1 -15555.742,E2 -15555.742} C_VEL
LIN {X 0,Y 312.695,Z 688.752,A -85,B 0,C 180,E1 -15557.671,E2 -15557.671} C_VEL
LIN {X 0,Y 311.916,Z 694.812,A -85,B 0,C 180,E1 -15559.615,E2 -15559.615} C_VEL
LIN {X 0,Y 311.288,Z 699.595,A -85,B 0,C 180,E1 -15561.561,E2 -15561.561} C_VEL
LIN {X 0,Y 310.981,Z 703.246,A -85,B 0,C 180,E1 -15563.512,E2 -15563.512} C_VEL
LIN {X 0,Y 310.841,Z 705.126,A -85,B 0,C 180,E1 -15564.811,E2 -15564.811} C_VEL
LIN {X 0,Y 310.787,Z 706.544,A -85,B 0,C 180,E1 -15566.11,E2 -15566.11} C_VEL
LIN {X 0,Y 310.735,Z 707.544,A -85,B 0,C 180,E1 -15567.407,E2 -15567.407} C_VEL
LIN {X 0,Y 310.68,Z 708.154,A -85,B 0,C 180,E1 -15568.704,E2 -15568.704} C_VEL
LIN {X 0,Y 310.703,Z 708.371,A -85,B 0,C 180,E1 -15570,E2 -15570} C_VEL
LIN {X 0,Y 310.712,Z 708.148,A -85,B 0,C 180,E1 -15571.296,E2 -15571.296} C_VEL
LIN {X 0,Y 310.74,Z 707.533,A -85,B 0,C 180,E1 -15572.592,E2 -15572.592} C_VEL
LIN {X 0,Y 310.81,Z 706.529,A -85,B 0,C 180,E1 -15573.89,E2 -15573.89} C_VEL
LIN {X 0,Y 310.912,Z 704.051,A -85,B 0,C 180,E1 -15575.957,E2 -15575.957} C_VEL
LIN {X 0,Y 311.17,Z 700.902,A -85,B 0,C 180,E1 -15577.788,E2 -15577.788} C_VEL
LIN {X 0,Y 311.697,Z 696.504,A -85,B 0,C 180,E1 -15579.736,E2 -15579.736} C_VEL
LIN {X 0,Y 312.578,Z 689.804,A -85,B 0,C 180,E1 -15582.004,E2 -15582.004} C_VEL
LIN {X 0,Y 313.692,Z 682.481,A -85,B 0,C 180,E1 -15583.936,E2 -15583.936} C_VEL
LIN {X 0,Y 315.002,Z 673.474,A -85,B 0,C 180,E1 -15585.836,E2 -15585.836} C_VEL
LIN {X 0,Y 316.345,Z 663.821,A -85,B 0,C 180,E1 -15587.452,E2 -15587.452} C_VEL
LIN {X 0,Y 317.764,Z 653.247,A -85,B 0,C 180,E1 -15588.872,E2 -15588.872} C_VEL
LIN {X 0,Y 319.041,Z 642.997,A -85,B 0,C 180,E1 -15589.965,E2 -15589.965} C_VEL
LIN {X 0,Y 320.291,Z 630.677,A -85,B 0,C 180,E1 -15590.974,E2 -15590.974} C_VEL
LIN {X 0,Y 321.316,Z 617.741,A -85,B 0,C 180,E1 -15591.744,E2 -15591.744} C_VEL
LIN {X 0,Y 321.78,Z 614.875,A -85,B 0,C 180,E1 -15591.964,E2 -15591.964} C_VEL
LIN {X 0,Y 324.329,Z 602.642,A -85,B 0,C 180,E1 -15593.126,E2 -15593.126} C_VEL
LIN {X 0,Y 326.751,Z 589.274,A -85,B 0,C 180,E1 -15594.121,E2 -15594.121} C_VEL
LIN {X 0,Y 328.748,Z 574.812,A -85,B 0,C 180,E1 -15594.932,E2 -15594.932} C_VEL
LIN {X 0,Y 330.224,Z 559.403,A -85,B 0,C 180,E1 -15595.561,E2 -15595.561} C_VEL
LIN {X 0,Y 332.681,Z 527.601,A -85,B 0,C 180,E1 -15596.717,E2 -15596.717} C_VEL
LIN {X 0,Y 332.564,Z 510.067,A -85,B 0,C 180,E1 -15597.631,E2 -15597.631} C_VEL
LIN {X 0,Y 331.609,Z 494.309,A -85,B 0,C 180,E1 -15598.654,E2 -15598.654} C_VEL
LIN {X 0,Y 329.955,Z 479.092,A -85,B 0,C 180,E1 -15599.861,E2 -15599.861} C_VEL
LIN {X 0,Y 327.817,Z 463.931,A -85,B 0,C 180,E1 -15601.284,E2 -15601.284} C_VEL
LIN {X 0,Y 325.956,Z 453.168,A -85,B 0,C 180,E1 -15602.477,E2 -15602.477} C_VEL
LIN {X 0,Y 323.598,Z 446.646,A -85,B 0,C 180,E1 -15603.722,E2 -15603.722} C_VEL
LIN {X 0,Y 322.22,Z 439.912,A -85,B 0,C 180,E1 -15606.195,E2 -15606.195} C_VEL
LIN {X 0,Y 320.793,Z 434.388,A -85,B 0,C 180,E1 -15608.636,E2 -15608.636} C_VEL
LIN {X 0,Y 319.182,Z 428.995,A -85,B 0,C 180,E1 -15611.527,E2 -15611.527} C_VEL
LIN {X 0,Y 317.557,Z 424.248,A -85,B 0,C 180,E1 -15614.911,E2 -15614.911} C_VEL
LIN {X 0,Y 316.442,Z 421.025,A -85,B 0,C 180,E1 -15618.219,E2 -15618.219} C_VEL
LIN {X 0,Y 315.794,Z 419.158,A -85,B 0,C 180,E1 -15621.454,E2 -15621.454} C_VEL
LIN {X 0,Y 315.756,Z 418.802,A -85,B 0,C 180,E1 -15623.252,E2 -15623.252} C_VEL
LIN {X 0,Y 318.589,Z 421.171,A -85,B 0,C 180,E1 -15625.179,E2 -15625.179} C_VEL
LIN {X 0,Y 320.21,Z 422.556,A -85,B 0,C 180,E1 -15626.023,E2 -15626.023} C_VEL
LIN {X 0,Y 323.208,Z 425.336,A -85,B 0,C 180,E1 -15627.451,E2 -15627.451} C_VEL
LIN {X 0,Y 325.879,Z 428.161,A -85,B 0,C 180,E1 -15628.563,E2 -15628.563} C_VEL
LIN {X 0,Y 327.964,Z 431.065,A -85,B 0,C 180,E1 -15629.416,E2 -15629.416} C_VEL
LIN {X 0,Y 331.062,Z 436.085,A -85,B 0,C 180,E1 -15630.593,E2 -15630.593} C_VEL
LIN {X 0,Y 334.324,Z 441.458,A -85,B 0,C 180,E1 -15631.713,E2 -15631.713} C_VEL
LIN {X 0,Y 338.098,Z 449.002,A -85,B 0,C 180,E1 -15632.967,E2 -15632.967} C_VEL
LIN {X 0,Y 334.371,Z 489.309,A -85,B 0,C 180,E1 -15634.52,E2 -15634.52} C_VEL
LIN {X 0,Y 333.278,Z 508.516,A -85,B 0,C 180,E1 -15635.376,E2 -15635.376} C_VEL
LIN {X 0,Y 332.282,Z 521.2,A -85,B 0,C 180,E1 -15636.165,E2 -15636.165} C_VEL
LIN {X 0,Y 331.093,Z 531.979,A -85,B 0,C 180,E1 -15637.043,E2 -15637.043} C_VEL
LIN {X 0,Y 329.239,Z 545.042,A -85,B 0,C 180,E1 -15638.394,E2 -15638.394} C_VEL
LIN {X 0,Y 327.146,Z 556.476,A -85,B 0,C 180,E1 -15639.896,E2 -15639.896} C_VEL
LIN {X 0,Y 325.296,Z 565.602,A -85,B 0,C 180,E1 -15641.417,E2 -15641.417} C_VEL
LIN {X 0,Y 323.198,Z 574.31,A -85,B 0,C 180,E1 -15643.216,E2 -15643.216} C_VEL
LIN {X 0,Y 321.185,Z 581.631,A -85,B 0,C 180,E1 -15645.102,E2 -15645.102} C_VEL
LIN {X 0,Y 319.165,Z 588.041,A -85,B 0,C 180,E1 -15647.279,E2 -15647.279} C_VEL
LIN {X 0,Y 317.686,Z 592.193,A -85,B 0,C 180,E1 -15649.162,E2 -15649.162} C_VEL
LIN {X 0,Y 316.365,Z 595.272,A -85,B 0,C 180,E1 -15651.054,E2 -15651.054} C_VEL
LIN {X 0,Y 315.566,Z 596.745,A -85,B 0,C 180,E1 -15652.321,E2 -15652.321} C_VEL
LIN {X 0,Y 314.969,Z 597.716,A -85,B 0,C 180,E1 -15653.594,E2 -15653.594} C_VEL
LIN {X 0,Y 314.542,Z 598.258,A -85,B 0,C 180,E1 -15654.872,E2 -15654.872} C_VEL
LIN {X 0,Y 314.087,Z 598.402,A -85,B 0,C 180,E1 -15656.151,E2 -15656.151} C_VEL
LIN {X 0,Y 313.622,Z 598.092,A -85,B 0,C 180,E1 -15657.431,E2 -15657.431} C_VEL
LIN {X 0,Y 313.302,Z 597.356,A -85,B 0,C 180,E1 -15658.715,E2 -15658.715} C_VEL
LIN {X 0,Y 312.895,Z 596.227,A -85,B 0,C 180,E1 -15660,E2 -15660} C_VEL
LIN {X 0,Y 312.817,Z 593.621,A -85,B 0,C 180,E1 -15661.931,E2 -15661.931} C_VEL
LIN {X 0,Y 312.684,Z 589.998,A -85,B 0,C 180,E1 -15663.866,E2 -15663.866} C_VEL
LIN {X 0,Y 312.863,Z 585.224,A -85,B 0,C 180,E1 -15665.802,E2 -15665.802} C_VEL
LIN {X 0,Y 313.146,Z 579.184,A -85,B 0,C 180,E1 -15667.739,E2 -15667.739} C_VEL
LIN {X 0,Y 313.619,Z 571.347,A -85,B 0,C 180,E1 -15669.76,E2 -15669.76} C_VEL
LIN {X 0,Y 314.08,Z 562.391,A -85,B 0,C 180,E1 -15671.618,E2 -15671.618} C_VEL
LIN {X 0,Y 314.701,Z 551.802,A -85,B 0,C 180,E1 -15673.397,E2 -15673.397} C_VEL
LIN {X 0,Y 315.299,Z 541.127,A -85,B 0,C 180,E1 -15674.853,E2 -15674.853} C_VEL
LIN {X 0,Y 315.953,Z 529.412,A -85,B 0,C 180,E1 -15676.144,E2 -15676.144} C_VEL
LIN {X 0,Y 316.459,Z 516.627,A -85,B 0,C 180,E1 -15677.262,E2 -15677.262} C_VEL
LIN {X 0,Y 316.898,Z 502.758,A -85,B 0,C 180,E1 -15678.172,E2 -15678.172} C_VEL
LIN {X 0,Y 317.205,Z 489.559,A -85,B 0,C 180,E1 -15678.781,E2 -15678.781} C_VEL
LIN {X 0,Y 317.981,Z 449.168,A -85,B 0,C 180,E1 -15680.078,E2 -15680.078} C_VEL
LIN {X 0,Y 318.504,Z 429.235,A -85,B 0,C 180,E1 -15680.72,E2 -15680.72} C_VEL
LIN {X 0,Y 312.77,Z 410.456,A -85,B 0,C 180,E1 -15681.604,E2 -15681.604} C_VEL
LIN {X 0,Y 312.583,Z 409.614,A -85,B 0,C 180,E1 -15681.864,E2 -15681.864} C_VEL
LIN {X 0,Y 312.535,Z 409.554,A -85,B 0,C 180,E1 -15685.909,E2 -15685.909} C_VEL
LIN {X 0,Y 312.502,Z 409.544,A -85,B 0,C 180,E1 -15689.655,E2 -15689.655} C_VEL
LIN {X 0,Y 312.521,Z 409.539,A -85,B 0,C 180,E1 -15693.689,E2 -15693.689} C_VEL
LIN {X 0,Y 312.522,Z 409.548,A -85,B 0,C 180,E1 -15697.386,E2 -15697.386} C_VEL
LIN {X 0,Y 312.491,Z 409.559,A -85,B 0,C 180,E1 -15700.709,E2 -15700.709} C_VEL
LIN {X 0,Y 312.453,Z 409.564,A -85,B 0,C 180,E1 -15704.21,E2 -15704.21} C_VEL
LIN {X 0,Y 312.485,Z 409.555,A -85,B 0,C 180,E1 -15707.919,E2 -15707.919} C_VEL
